METHOD bitXIsEqualTo
VAR_INPUT
	(* current value to check *)
	currentValue	:WORD;
	(* number of bit to check *)
	number			:BitNumberWord;
	(* expected value of bit *)
	expectedValue	:BOOL;
	(* message if the assertion is false *)
	message			:AssertMessage;
END_VAR
IF (
	TO_BOOL(
		TO_WORD(SHL(THIS^.LSB, number))
		AND currentValue
	) <> expectedValue
) THEN
	THIS^.assertionWasWrong(message, THIS^.getDebugInfo('bitXIsEqualTo'));
END_IF
END_METHOD

(*

short summary
=================
This assertion method checks if the selected bit of current value
is not equal to the unexpected value

.. <legal notes>

legal notes
=================
| SPDX-FileCopyrightText: © 2022 ekvip automation GmbH <info@ekvip.de>
| SPDX-License-Identifier: Apache-2.0
| For details check: Apache-2.0_

.. _Apache-2.0: https://www.apache.org/licenses/LICENSE-2.0

.. </legal notes>

parameters
=================

*)

METHOD bitXIsNotEqualTo
VAR_INPUT
	(* current value to check *)
	currentValue	:WORD;
	(* number of bit to check *)
	number			:BitNumberWord;
	(* unexpected value of bit *)
	unexpectedValue	:BOOL;
	(* message if the assertion is false *)
	message			:AssertMessage;
END_VAR
IF (
	TO_BOOL(
		TO_WORD(SHL(THIS^.LSB, number))
		AND currentValue
	) = unexpectedValue
) THEN
	THIS^.assertionWasWrong(message, THIS^.getDebugInfo('bitXIsNotEqualTo'));
END_IF
END_METHOD

(*

short summary
=================
This assertion method checks if the selected bit of current value
is set

.. <legal notes>

legal notes
=================
| SPDX-FileCopyrightText: © 2022 ekvip automation GmbH <info@ekvip.de>
| SPDX-License-Identifier: Apache-2.0
| For details check: Apache-2.0_

.. _Apache-2.0: https://www.apache.org/licenses/LICENSE-2.0

.. </legal notes>

parameters
=================

*)

METHOD bitXIsSet
VAR_INPUT
	(* current value to check *)
	currentValue	:WORD;
	(* number of bit to check *)
	number			:BitNumberWord;
	(* message if the assertion is false *)
	message			:AssertMessage;
END_VAR
IF (
	NOT TO_BOOL(
		TO_WORD(SHL(THIS^.LSB, number))
		AND currentValue
	)
) THEN
	THIS^.assertionWasWrong(message, THIS^.getDebugInfo('bitXIsSet'));
END_IF
END_METHOD

(*

short summary
=================
This assertion method checks if the selected bit of current value
is unset

.. <legal notes>

legal notes
=================
| SPDX-FileCopyrightText: © 2022 ekvip automation GmbH <info@ekvip.de>
| SPDX-License-Identifier: Apache-2.0
| For details check: Apache-2.0_

.. _Apache-2.0: https://www.apache.org/licenses/LICENSE-2.0

.. </legal notes>

parameters
=================

*)

METHOD bitXIsUnset
VAR_INPUT
	(* current value to check *)
	currentValue	:WORD;
	(* number of bit to check *)
	number			:BitNumberWord;
	(* message if the assertion is false *)
	message			:AssertMessage;
END_VAR
IF (
	TO_BOOL(
		TO_WORD(SHL(THIS^.LSB, number))
		AND currentValue
	)
) THEN
	THIS^.assertionWasWrong(message, THIS^.getDebugInfo('bitXIsUnset'));
END_IF
END_METHOD

(*

short summary
=================
This abstract property returns the class name of the concrete object, 
It's for debugging purpose

.. <legal notes>

legal notes
=================
| SPDX-FileCopyrightText: © 2022 ekvip automation GmbH <info@ekvip.de>
| SPDX-License-Identifier: Apache-2.0
| For details check: Apache-2.0_

.. _Apache-2.0: https://www.apache.org/licenses/LICENSE-2.0

.. </legal notes>

*)

PROPERTY className :CNM_AbstractObject.ClassName
GET
className := 'CNM_AssertionInterfaceLib.WordAssertions';
END_GET
END_PROPERTY

(*

short summary
=================
This assertion method checks if the least significant bit of current value
is equal to the expected value

.. <legal notes>

legal notes
=================
| SPDX-FileCopyrightText: © 2022 ekvip automation GmbH <info@ekvip.de>
| SPDX-License-Identifier: Apache-2.0
| For details check: Apache-2.0_

.. _Apache-2.0: https://www.apache.org/licenses/LICENSE-2.0

.. </legal notes>

parameters
=================

*)

METHOD lsbIsEqualTo
VAR_INPUT
	(* current value to check *)
	currentValue	:WORD;
	(* expected value of lsb *)
	expectedValue	:BOOL;
	(* message if the assertion is false *)
	message			:AssertMessage;
END_VAR
IF (TO_BOOL(currentValue AND THIS^.LSB) <> expectedValue) THEN
	THIS^.assertionWasWrong(message, THIS^.getDebugInfo('lsbIsEqualTo'));
END_IF
END_METHOD

(*

short summary
=================
This assertion method checks if the least significant bit of current value
is not equal to the unexpected value

.. <legal notes>

legal notes
=================
| SPDX-FileCopyrightText: © 2022 ekvip automation GmbH <info@ekvip.de>
| SPDX-License-Identifier: Apache-2.0
| For details check: Apache-2.0_

.. _Apache-2.0: https://www.apache.org/licenses/LICENSE-2.0

.. </legal notes>

parameters
=================

*)

METHOD lsbIsNotEqualTo
VAR_INPUT
	(* current value to check *)
	currentValue	:WORD;
	(* unexpected value of lsb *)
	unexpectedValue	:BOOL;
	(* message if the assertion is false *)
	message			:AssertMessage;
END_VAR
IF (TO_BOOL(currentValue AND THIS^.LSB) = unexpectedValue) THEN
	THIS^.assertionWasWrong(message, THIS^.getDebugInfo('lsbIsNotEqualTo'));
END_IF
END_METHOD

(*

short summary
=================
This assertion method checks if the least significant bit of current value
is set

.. <legal notes>

legal notes
=================
| SPDX-FileCopyrightText: © 2022 ekvip automation GmbH <info@ekvip.de>
| SPDX-License-Identifier: Apache-2.0
| For details check: Apache-2.0_

.. _Apache-2.0: https://www.apache.org/licenses/LICENSE-2.0

.. </legal notes>

parameters
=================

*)

METHOD lsbIsSet
VAR_INPUT
	(* current value to check *)
	currentValue	:WORD;
	(* message if the assertion is false *)
	message			:AssertMessage;
END_VAR
IF (NOT TO_BOOL(currentValue AND THIS^.LSB)) THEN
	THIS^.assertionWasWrong(message, THIS^.getDebugInfo('lsbIsSet'));
END_IF
END_METHOD

(*

short summary
=================
This assertion method checks if the least significant bit of current value
is unset

.. <legal notes>

legal notes
=================
| SPDX-FileCopyrightText: © 2022 ekvip automation GmbH <info@ekvip.de>
| SPDX-License-Identifier: Apache-2.0
| For details check: Apache-2.0_

.. _Apache-2.0: https://www.apache.org/licenses/LICENSE-2.0

.. </legal notes>

parameters
=================

*)

METHOD lsbIsUnset
VAR_INPUT
	(* current value to check *)
	currentValue	:WORD;
	(* message if the assertion is false *)
	message			:AssertMessage;
END_VAR
IF (TO_BOOL(currentValue AND THIS^.LSB)) THEN
	THIS^.assertionWasWrong(message, THIS^.getDebugInfo('lsbIsUnset'));
END_IF
END_METHOD

(*

short summary
=================
This assertion method checks if the most significant bit of current value
is equal to the expected value

.. <legal notes>

legal notes
=================
| SPDX-FileCopyrightText: © 2022 ekvip automation GmbH <info@ekvip.de>
| SPDX-License-Identifier: Apache-2.0
| For details check: Apache-2.0_

.. _Apache-2.0: https://www.apache.org/licenses/LICENSE-2.0

.. </legal notes>

parameters
=================

*)

METHOD msbIsEqualTo
VAR_INPUT
	(* current value to check *)
	currentValue	:WORD;
	(* expected value of msb *)
	expectedValue	:BOOL;
	(* message if the assertion is false *)
	message			:AssertMessage;
END_VAR
IF (TO_BOOL(currentValue AND THIS^.MSB) <> expectedValue) THEN
	THIS^.assertionWasWrong(message, THIS^.getDebugInfo('msbIsEqualTo'));
END_IF
END_METHOD

(*

short summary
=================
This assertion method checks if the most significant bit of current value
is not equal to the unexpected value

.. <legal notes>

legal notes
=================
| SPDX-FileCopyrightText: © 2022 ekvip automation GmbH <info@ekvip.de>
| SPDX-License-Identifier: Apache-2.0
| For details check: Apache-2.0_

.. _Apache-2.0: https://www.apache.org/licenses/LICENSE-2.0

.. </legal notes>

parameters
=================

*)

METHOD msbIsNotEqualTo
VAR_INPUT
	(* current value to check *)
	currentValue	:WORD;
	(* unexpected value of msb *)
	unexpectedValue	:BOOL;
	(* message if the assertion is false *)
	message			:AssertMessage;
END_VAR
IF (TO_BOOL(currentValue AND THIS^.MSB) = unexpectedValue) THEN
	THIS^.assertionWasWrong(message, THIS^.getDebugInfo('msbIsNotEqualTo'));
END_IF
END_METHOD

(*

short summary
=================
This assertion method checks if the most significant bit of current value
is set

.. <legal notes>

legal notes
=================
| SPDX-FileCopyrightText: © 2022 ekvip automation GmbH <info@ekvip.de>
| SPDX-License-Identifier: Apache-2.0
| For details check: Apache-2.0_

.. _Apache-2.0: https://www.apache.org/licenses/LICENSE-2.0

.. </legal notes>

parameters
=================

*)

METHOD msbIsSet
VAR_INPUT
	(* current value to check *)
	currentValue	:WORD;
	(* message if the assertion is false *)
	message			:AssertMessage;
END_VAR
IF (NOT TO_BOOL(currentValue AND THIS^.MSB)) THEN
	THIS^.assertionWasWrong(message, THIS^.getDebugInfo('msbIsSet'));
END_IF
END_METHOD

(*

short summary
=================
This assertion method checks if the most significant bit of current value
is unset

.. <legal notes>

legal notes
=================
| SPDX-FileCopyrightText: © 2022 ekvip automation GmbH <info@ekvip.de>
| SPDX-License-Identifier: Apache-2.0
| For details check: Apache-2.0_

.. _Apache-2.0: https://www.apache.org/licenses/LICENSE-2.0

.. </legal notes>

parameters
=================

*)

METHOD msbIsUnset
VAR_INPUT
	(* current value to check *)
	currentValue	:WORD;
	(* message if the assertion is false *)
	message			:AssertMessage;
END_VAR
IF (TO_BOOL(currentValue AND THIS^.MSB)) THEN
	THIS^.assertionWasWrong(message, THIS^.getDebugInfo('msbIsUnset'));
END_IF
END_METHOD

(*

short summary
=================
This assertion method checks if the result current value bitwise ``OR`` mask is equal to the expected value

.. <legal notes>

legal notes
=================
| SPDX-FileCopyrightText: © 2022 ekvip automation GmbH <info@ekvip.de>
| SPDX-License-Identifier: Apache-2.0
| For details check: Apache-2.0_

.. _Apache-2.0: https://www.apache.org/licenses/LICENSE-2.0

.. </legal notes>

parameters
=================

*)

METHOD orMaskIsEqualTo
VAR_INPUT
	(* current value to check *)
	currentValue	:WORD;
	(* 2nd operand for bitwise operation *)
	mask			:WORD;
	(* expected result after masking *)
	expectedValue	:WORD;
	(* message if the assertion is false *)
	message			:AssertMessage;
END_VAR
IF ((currentValue OR mask) <> expectedValue) THEN
	THIS^.assertionWasWrong(message, THIS^.getDebugInfo('orMaskIsEqualTo'));
END_IF
END_METHOD

(*

short summary
=================
This assertion method checks if the result current value bitwise ``OR`` mask 
is not equal to the unexpected value

.. <legal notes>

legal notes
=================
| SPDX-FileCopyrightText: © 2022 ekvip automation GmbH <info@ekvip.de>
| SPDX-License-Identifier: Apache-2.0
| For details check: Apache-2.0_

.. _Apache-2.0: https://www.apache.org/licenses/LICENSE-2.0

.. </legal notes>

parameters
=================

*)

METHOD orMaskIsNotEqualTo
VAR_INPUT
	(* current value to check *)
	currentValue	:WORD;
	(* 2nd operand for bitwise operation *)
	mask			:WORD;
	(* unexpected result after masking *)
	unexpectedValue	:WORD;
	(* message if the assertion is false *)
	message			:AssertMessage;
END_VAR
IF ((currentValue OR mask) = unexpectedValue) THEN
	THIS^.assertionWasWrong(message, THIS^.getDebugInfo('orMaskIsNotEqualTo'));
END_IF
END_METHOD

(*

short summary
=================
This assertion method checks if the current value is equal to the expected value

.. <legal notes>

legal notes
=================
| SPDX-FileCopyrightText: © 2022 ekvip automation GmbH <info@ekvip.de>
| SPDX-License-Identifier: Apache-2.0
| For details check: Apache-2.0_

.. _Apache-2.0: https://www.apache.org/licenses/LICENSE-2.0

.. </legal notes>

parameters
=================

*)

METHOD valueIsEqualTo
VAR_INPUT
	(* current value to check *)
	currentValue	:WORD;
	(* expected value to compare *)
	expectedValue	:WORD;
	(* message if the assertion is false *)
	message			:AssertMessage;
END_VAR
IF (currentValue <> expectedValue) THEN
	THIS^.assertionWasWrong(message, THIS^.getDebugInfo('valueIsEqualTo'));
END_IF
END_METHOD

(*

short summary
=================
This assertion method checks if the current value is greater than the less value

.. <legal notes>

legal notes
=================
| SPDX-FileCopyrightText: © 2022 ekvip automation GmbH <info@ekvip.de>
| SPDX-License-Identifier: Apache-2.0
| For details check: Apache-2.0_

.. _Apache-2.0: https://www.apache.org/licenses/LICENSE-2.0

.. </legal notes>

parameters
=================

*)

METHOD valueIsGreaterThan
VAR_INPUT
	(* current value to check *)
	currentValue	:WORD;
	(* less than lower limit *)
	lessValue		:WORD;
	(* message if the assertion is false *)
	message			:AssertMessage;
END_VAR
IF (currentValue <= lessValue) THEN
	THIS^.assertionWasWrong(message, THIS^.getDebugInfo('valueIsGreaterThan'));
END_IF
END_METHOD

(*

short summary
=================
This assertion method checks if the current value is inside a limit

.. attention:: 
	limits are included: ``valueIsInRangeOf(3, 3, 3)`` is a true assertion

.. <legal notes>

legal notes
=================
| SPDX-FileCopyrightText: © 2022 ekvip automation GmbH <info@ekvip.de>
| SPDX-License-Identifier: Apache-2.0
| For details check: Apache-2.0_

.. _Apache-2.0: https://www.apache.org/licenses/LICENSE-2.0

.. </legal notes>

parameters
=================

*)

METHOD valueIsInRangeOf
VAR_INPUT
	(* lower limit for the current value *)
	lowerLimit		:WORD;
	(* current value to check *)
	currentValue	:WORD;
	(* upper limit for the current value *)
	upperLimit		:WORD;
	(* message if the assertion is false *)
	message			:AssertMessage;
END_VAR
IF (
	(currentValue < lowerLimit)
	OR (currentValue > upperLimit)
) THEN
	THIS^.assertionWasWrong(message, THIS^.getDebugInfo('valueIsInRangeOf'));
END_IF
END_METHOD

(*

short summary
=================
This assertion method checks if the current value is less than the greater value

.. <legal notes>

legal notes
=================
| SPDX-FileCopyrightText: © 2022 ekvip automation GmbH <info@ekvip.de>
| SPDX-License-Identifier: Apache-2.0
| For details check: Apache-2.0_

.. _Apache-2.0: https://www.apache.org/licenses/LICENSE-2.0

.. </legal notes>

parameters
=================

*)

METHOD valueIsLessThan
VAR_INPUT
	(* current value to check *)
	currentValue	:WORD;
	(* greater than upper limit *)
	greaterValue	:WORD;
	(* message if the assertion is false *)
	message			:AssertMessage;
END_VAR
IF (currentValue >= greaterValue) THEN
	THIS^.assertionWasWrong(message, THIS^.getDebugInfo('valueIsLessThan'));
END_IF
END_METHOD

(*

short summary
=================
This assertion method checks if the current value is less than or equal to the maximum value

.. <legal notes>

legal notes
=================
| SPDX-FileCopyrightText: © 2022 ekvip automation GmbH <info@ekvip.de>
| SPDX-License-Identifier: Apache-2.0
| For details check: Apache-2.0_

.. _Apache-2.0: https://www.apache.org/licenses/LICENSE-2.0

.. </legal notes>

parameters
=================

*)

METHOD valueIsMax
VAR_INPUT
	(* current value to check *)
	currentValue	:WORD;
	(* upper limit for the current value *)
	maximumValue	:WORD;
	(* message if the assertion is false *)
	message			:AssertMessage;
END_VAR
IF (currentValue > maximumValue) THEN
	THIS^.assertionWasWrong(message, THIS^.getDebugInfo('valueIsMax'));
END_IF
END_METHOD

(*

short summary
=================
This assertion method checks if the current value is greater than or equal to the minimum value

.. <legal notes>

legal notes
=================
| SPDX-FileCopyrightText: © 2022 ekvip automation GmbH <info@ekvip.de>
| SPDX-License-Identifier: Apache-2.0
| For details check: Apache-2.0_

.. _Apache-2.0: https://www.apache.org/licenses/LICENSE-2.0

.. </legal notes>

parameters
=================

*)

METHOD valueIsMin
VAR_INPUT
	(* current value to check *)
	currentValue	:WORD;
	(* lower limit for the current value *)
	minimumValue	:WORD;
	(* message if the assertion is false *)
	message			:AssertMessage;
END_VAR
IF (currentValue < minimumValue) THEN
	THIS^.assertionWasWrong(message, THIS^.getDebugInfo('valueIsMin'));
END_IF
END_METHOD

(*

short summary
=================
This assertion method checks if the current value is not equal to the unexpected value

.. <legal notes>

legal notes
=================
| SPDX-FileCopyrightText: © 2022 ekvip automation GmbH <info@ekvip.de>
| SPDX-License-Identifier: Apache-2.0
| For details check: Apache-2.0_

.. _Apache-2.0: https://www.apache.org/licenses/LICENSE-2.0

.. </legal notes>

parameters
=================

*)

METHOD valueIsNotEqualTo
VAR_INPUT
	(* current value to check *)
	currentValue	:WORD;
	(* unexpected value to compare *)
	unexpectedValue	:WORD;
	(* message if the assertion is false *)
	message			:AssertMessage;
END_VAR
IF (currentValue = unexpectedValue) THEN
	THIS^.assertionWasWrong(message, THIS^.getDebugInfo('valueIsNotEqualTo'));
END_IF
END_METHOD

(*

short summary
=================
This assertion method checks if the result current value bitwise ``XOR`` mask is equal to the expected value

.. <legal notes>

legal notes
=================
| SPDX-FileCopyrightText: © 2022 ekvip automation GmbH <info@ekvip.de>
| SPDX-License-Identifier: Apache-2.0
| For details check: Apache-2.0_

.. _Apache-2.0: https://www.apache.org/licenses/LICENSE-2.0

.. </legal notes>

parameters
=================

*)

METHOD xorMaskIsEqualTo
VAR_INPUT
	(* current value to check *)
	currentValue	:WORD;
	(* 2nd operand for bitwise operation *)
	mask			:WORD;
	(* expected result after masking *)
	expectedValue	:WORD;
	(* message if the assertion is false *)
	message			:AssertMessage;
END_VAR
IF ((currentValue XOR mask) <> expectedValue) THEN
	THIS^.assertionWasWrong(message, THIS^.getDebugInfo('xorMaskIsEqualTo'));
END_IF
END_METHOD

(*

short summary
=================
This assertion method checks if the result current value bitwise ``XOR`` mask 
is not equal to the unexpected value

.. <legal notes>

legal notes
=================
| SPDX-FileCopyrightText: © 2022 ekvip automation GmbH <info@ekvip.de>
| SPDX-License-Identifier: Apache-2.0
| For details check: Apache-2.0_

.. _Apache-2.0: https://www.apache.org/licenses/LICENSE-2.0

.. </legal notes>

parameters
=================

*)

METHOD xorMaskIsNotEqualTo
VAR_INPUT
	(* current value to check *)
	currentValue	:WORD;
	(* 2nd operand for bitwise operation *)
	mask			:WORD;
	(* unexpected result after masking *)
	unexpectedValue	:WORD;
	(* message if the assertion is false *)
	message			:AssertMessage;
END_VAR
IF ((currentValue XOR mask) = unexpectedValue) THEN
	THIS^.assertionWasWrong(message, THIS^.getDebugInfo('xorMaskIsNotEqualTo'));
END_IF
END_METHOD

END_FUNCTION_BLOCK

// ---- Assertor/Assertions/BitNumberAssertions/Dword/classes/DWordAssertions.TcPOU
(*

short summary
=================
This class provides assert statements for double words  
It implements :ref:`IDWordAssertions`

.. <legal notes>

legal notes
=================
| SPDX-FileCopyrightText: © 2022 ekvip automation GmbH <info@ekvip.de>
| SPDX-License-Identifier: Apache-2.0
| For details check: Apache-2.0_

.. _Apache-2.0: https://www.apache.org/licenses/LICENSE-2.0

.. </legal notes>

methods and properties
=======================

*)

{attribute 'reflection'}
FUNCTION_BLOCK INTERNAL DWordAssertions EXTENDS AbstactAssertion IMPLEMENTS IDWordAssertions
VAR
END_VAR
VAR CONSTANT
	(* least significant bit *)
	LSB	:DWORD := 16#0000_0001;
	(* most significant bit *)
	MSB :DWORD := 16#8000_0000;
END_VAR

(*

short summary
=================
This assertion method checks if the result current value bitwise ``AND`` mask is equal to the expected value

.. <legal notes>

legal notes
=================
| SPDX-FileCopyrightText: © 2022 ekvip automation GmbH <info@ekvip.de>
| SPDX-License-Identifier: Apache-2.0
| For details check: Apache-2.0_

.. _Apache-2.0: https://www.apache.org/licenses/LICENSE-2.0

.. </legal notes>

parameters
=================

*)

METHOD andMaskIsEqualTo
VAR_INPUT
	(* current value to check *)
	currentValue	:DWORD;
	(* 2nd operand for bitwise operation *)
	mask			:DWORD;
	(* expected result after masking *)
	expectedValue	:DWORD;
	(* message if the assertion is false *)
	message			:AssertMessage;
END_VAR
IF ((currentValue AND mask) <> expectedValue) THEN
	THIS^.assertionWasWrong(message, THIS^.getDebugInfo('andMaskIsEqualTo'));
END_IF
END_METHOD

(*

short summary
=================
This assertion method checks if the result current value bitwise ``AND`` mask
is not equal to the unexpected value

.. <legal notes>

legal notes
=================
| SPDX-FileCopyrightText: © 2022 ekvip automation GmbH <info@ekvip.de>
| SPDX-License-Identifier: Apache-2.0
| For details check: Apache-2.0_

.. _Apache-2.0: https://www.apache.org/licenses/LICENSE-2.0

.. </legal notes>

parameters
=================

*)

METHOD andMaskIsNotEqualTo
VAR_INPUT
	(* current value to check *)
	currentValue	:DWORD;
	(* 2nd operand for bitwise operation *)
	mask			:DWORD;
	(* unexpected result after masking *)
	unexpectedValue	:DWORD;
	(* message if the assertion is false *)
	message			:AssertMessage;
END_VAR
IF ((currentValue AND mask) = unexpectedValue) THEN
	THIS^.assertionWasWrong(message, THIS^.getDebugInfo('andMaskIsNotEqualTo'));
END_IF
END_METHOD

(*

short summary
=================
This assertion method checks if the selected bit of current value
is equal to the expected value

.. <legal notes>

legal notes
=================
| SPDX-FileCopyrightText: © 2022 ekvip automation GmbH <info@ekvip.de>
| SPDX-License-Identifier: Apache-2.0
| For details check: Apache-2.0_

.. _Apache-2.0: https://www.apache.org/licenses/LICENSE-2.0

.. </legal notes>

parameters
=================

*)

METHOD bitXIsEqualTo
VAR_INPUT
	(* current value to check *)
	currentValue	:DWORD;
	(* number of bit to check *)
	number			:BitNumberDWord;
	(* expected value of bit *)
	expectedValue	:BOOL;
	(* message if the assertion is false *)
	message			:AssertMessage;
END_VAR
IF (
	TO_BOOL(
		TO_DWORD(SHL(THIS^.LSB, number))
		AND currentValue
	) <> expectedValue
) THEN
	THIS^.assertionWasWrong(message, THIS^.getDebugInfo('bitXIsEqualTo'));
END_IF
END_METHOD

(*

short summary
=================
This assertion method checks if the selected bit of current value
is not equal to the unexpected value

.. <legal notes>

legal notes
=================
| SPDX-FileCopyrightText: © 2022 ekvip automation GmbH <info@ekvip.de>
| SPDX-License-Identifier: Apache-2.0
| For details check: Apache-2.0_

.. _Apache-2.0: https://www.apache.org/licenses/LICENSE-2.0

.. </legal notes>

parameters
=================

*)

METHOD bitXIsNotEqualTo
VAR_INPUT
	(* current value to check *)
	currentValue	:DWORD;
	(* number of bit to check *)
	number			:BitNumberDWord;
	(* unexpected value of bit *)
	unexpectedValue	:BOOL;
	(* message if the assertion is false *)
	message			:AssertMessage;
END_VAR
IF (
	TO_BOOL(
		TO_DWORD(SHL(THIS^.LSB, number))
		AND currentValue
	) = unexpectedValue
) THEN
	THIS^.assertionWasWrong(message, THIS^.getDebugInfo('bitXIsNotEqualTo'));
END_IF
END_METHOD

(*

short summary
=================
This assertion method checks if the selected bit of current value
is set

.. <legal notes>

legal notes
=================
| SPDX-FileCopyrightText: © 2022 ekvip automation GmbH <info@ekvip.de>
| SPDX-License-Identifier: Apache-2.0
| For details check: Apache-2.0_

.. _Apache-2.0: https://www.apache.org/licenses/LICENSE-2.0

.. </legal notes>

parameters
=================

*)

METHOD bitXIsSet
VAR_INPUT
	(* current value to check *)
	currentValue	:DWORD;
	(* number of bit to check *)
	number			:BitNumberDWord;
	(* message if the assertion is false *)
	message			:AssertMessage;
END_VAR
IF (
	NOT TO_BOOL(
		TO_DWORD(SHL(THIS^.LSB, number))
		AND currentValue
	)
) THEN
	THIS^.assertionWasWrong(message, THIS^.getDebugInfo('bitXIsSet'));
END_IF
END_METHOD

(*

short summary
=================
This assertion method checks if the selected bit of current value
is unset

.. <legal notes>

legal notes
=================
| SPDX-FileCopyrightText: © 2022 ekvip automation GmbH <info@ekvip.de>
| SPDX-License-Identifier: Apache-2.0
| For details check: Apache-2.0_

.. _Apache-2.0: https://www.apache.org/licenses/LICENSE-2.0

.. </legal notes>

parameters
=================

*)

METHOD bitXIsUnset
VAR_INPUT
	(* current value to check *)
	currentValue	:DWORD;
	(* number of bit to check *)
	number			:BitNumberDWord;
	(* message if the assertion is false *)
	message			:AssertMessage;
END_VAR
IF (
	TO_BOOL(
		TO_DWORD(SHL(THIS^.LSB, number))
		AND currentValue
	)
) THEN
	THIS^.assertionWasWrong(message, THIS^.getDebugInfo('bitXIsUnset'));
END_IF
END_METHOD

(*

short summary
=================
This abstract property returns the class name of the concrete object, 
It's for debugging purpose

.. <legal notes>

legal notes
=================
| SPDX-FileCopyrightText: © 2022 ekvip automation GmbH <info@ekvip.de>
| SPDX-License-Identifier: Apache-2.0
| For details check: Apache-2.0_

.. _Apache-2.0: https://www.apache.org/licenses/LICENSE-2.0

.. </legal notes>

*)

PROPERTY className :CNM_AbstractObject.ClassName
GET
className := 'CNM_AssertionInterfaceLib.DWordAssertions';
END_GET
END_PROPERTY

(*

short summary
=================
This assertion method checks if the least significant bit of current value
is equal to the expected value

.. <legal notes>

legal notes
=================
| SPDX-FileCopyrightText: © 2022 ekvip automation GmbH <info@ekvip.de>
| SPDX-License-Identifier: Apache-2.0
| For details check: Apache-2.0_

.. _Apache-2.0: https://www.apache.org/licenses/LICENSE-2.0

.. </legal notes>

parameters
=================

*)

METHOD lsbIsEqualTo
VAR_INPUT
	(* current value to check *)
	currentValue	:DWORD;
	(* expected value of lsb *)
	expectedValue	:BOOL;
	(* message if the assertion is false *)
	message			:AssertMessage;
END_VAR
IF (TO_BOOL(currentValue AND THIS^.LSB) <> expectedValue) THEN
	THIS^.assertionWasWrong(message, THIS^.getDebugInfo('lsbIsEqualTo'));
END_IF
END_METHOD

(*

short summary
=================
This assertion method checks if the least significant bit of current value
is not equal to the unexpected value

.. <legal notes>

legal notes
=================
| SPDX-FileCopyrightText: © 2022 ekvip automation GmbH <info@ekvip.de>
| SPDX-License-Identifier: Apache-2.0
| For details check: Apache-2.0_

.. _Apache-2.0: https://www.apache.org/licenses/LICENSE-2.0

.. </legal notes>

parameters
=================

*)

METHOD lsbIsNotEqualTo
VAR_INPUT
	(* current value to check *)
	currentValue	:DWORD;
	(* unexpected value of lsb *)
	unexpectedValue	:BOOL;
	(* message if the assertion is false *)
	message			:AssertMessage;
END_VAR
IF (TO_BOOL(currentValue AND THIS^.LSB) = unexpectedValue) THEN
	THIS^.assertionWasWrong(message, THIS^.getDebugInfo('lsbIsNotEqualTo'));
END_IF
END_METHOD

(*

short summary
=================
This assertion method checks if the least significant bit of current value
is set

.. <legal notes>

legal notes
=================
| SPDX-FileCopyrightText: © 2022 ekvip automation GmbH <info@ekvip.de>
| SPDX-License-Identifier: Apache-2.0
| For details check: Apache-2.0_

.. _Apache-2.0: https://www.apache.org/licenses/LICENSE-2.0

.. </legal notes>

parameters
=================

*)

METHOD lsbIsSet
VAR_INPUT
	(* current value to check *)
	currentValue	:DWORD;
	(* message if the assertion is false *)
	message			:AssertMessage;
END_VAR
IF (NOT TO_BOOL(currentValue AND THIS^.LSB)) THEN
	THIS^.assertionWasWrong(message, THIS^.getDebugInfo('lsbIsSet'));
END_IF
END_METHOD

(*

short summary
=================
This assertion method checks if the least significant bit of current value
is unset

.. <legal notes>

legal notes
=================
| SPDX-FileCopyrightText: © 2022 ekvip automation GmbH <info@ekvip.de>
| SPDX-License-Identifier: Apache-2.0
| For details check: Apache-2.0_

.. _Apache-2.0: https://www.apache.org/licenses/LICENSE-2.0

.. </legal notes>

parameters
=================

*)

METHOD lsbIsUnset
VAR_INPUT
	(* current value to check *)
	currentValue	:DWORD;
	(* message if the assertion is false *)
	message			:AssertMessage;
END_VAR
IF (TO_BOOL(currentValue AND THIS^.LSB)) THEN
	THIS^.assertionWasWrong(message, THIS^.getDebugInfo('lsbIsUnset'));
END_IF
END_METHOD

(*

short summary
=================
This assertion method checks if the most significant bit of current value
is equal to the expected value

.. <legal notes>

legal notes
=================
| SPDX-FileCopyrightText: © 2022 ekvip automation GmbH <info@ekvip.de>
| SPDX-License-Identifier: Apache-2.0
| For details check: Apache-2.0_

.. _Apache-2.0: https://www.apache.org/licenses/LICENSE-2.0

.. </legal notes>

parameters
=================

*)

METHOD msbIsEqualTo
VAR_INPUT
	(* current value to check *)
	currentValue	:DWORD;
	(* expected value of msb *)
	expectedValue	:BOOL;
	(* message if the assertion is false *)
	message			:AssertMessage;
END_VAR
IF (TO_BOOL(currentValue AND THIS^.MSB) <> expectedValue) THEN
	THIS^.assertionWasWrong(message, THIS^.getDebugInfo('msbIsEqualTo'));
END_IF
END_METHOD

(*

short summary
=================
This assertion method checks if the most significant bit of current value
is not equal to the unexpected value

.. <legal notes>

legal notes
=================
| SPDX-FileCopyrightText: © 2022 ekvip automation GmbH <info@ekvip.de>
| SPDX-License-Identifier: Apache-2.0
| For details check: Apache-2.0_

.. _Apache-2.0: https://www.apache.org/licenses/LICENSE-2.0

.. </legal notes>

parameters
=================

*)

METHOD msbIsNotEqualTo
VAR_INPUT
	(* current value to check *)
	currentValue	:DWORD;
	(* unexpected value of msb *)
	unexpectedValue	:BOOL;
	(* message if the assertion is false *)
	message			:AssertMessage;
END_VAR
IF (TO_BOOL(currentValue AND THIS^.MSB) = unexpectedValue) THEN
	THIS^.assertionWasWrong(message, THIS^.getDebugInfo('msbIsNotEqualTo'));
END_IF
END_METHOD

(*

short summary
=================
This assertion method checks if the most significant bit of current value
is set

.. <legal notes>

legal notes
=================
| SPDX-FileCopyrightText: © 2022 ekvip automation GmbH <info@ekvip.de>
| SPDX-License-Identifier: Apache-2.0
| For details check: Apache-2.0_

.. _Apache-2.0: https://www.apache.org/licenses/LICENSE-2.0

.. </legal notes>

parameters
=================

*)

METHOD msbIsSet
VAR_INPUT
	(* current value to check *)
	currentValue	:DWORD;
	(* message if the assertion is false *)
	message			:AssertMessage;
END_VAR
IF (NOT TO_BOOL(currentValue AND THIS^.MSB)) THEN
	THIS^.assertionWasWrong(message, THIS^.getDebugInfo('msbIsSet'));
END_IF
END_METHOD

(*

short summary
=================
This assertion method checks if the most significant bit of current value
is unset

.. <legal notes>

legal notes
=================
| SPDX-FileCopyrightText: © 2022 ekvip automation GmbH <info@ekvip.de>
| SPDX-License-Identifier: Apache-2.0
| For details check: Apache-2.0_

.. _Apache-2.0: https://www.apache.org/licenses/LICENSE-2.0

.. </legal notes>

parameters
=================

*)

METHOD msbIsUnset
VAR_INPUT
	(* current value to check *)
	currentValue	:DWORD;
	(* message if the assertion is false *)
	message			:AssertMessage;
END_VAR
IF (TO_BOOL(currentValue AND THIS^.MSB)) THEN
	THIS^.assertionWasWrong(message, THIS^.getDebugInfo('msbIsUnset'));
END_IF
END_METHOD

(*

short summary
=================
This assertion method checks if the result current value bitwise ``OR`` mask is equal to the expected value

.. <legal notes>

legal notes
=================
| SPDX-FileCopyrightText: © 2022 ekvip automation GmbH <info@ekvip.de>
| SPDX-License-Identifier: Apache-2.0
| For details check: Apache-2.0_

.. _Apache-2.0: https://www.apache.org/licenses/LICENSE-2.0

.. </legal notes>

parameters
=================

*)

METHOD orMaskIsEqualTo
VAR_INPUT
	(* current value to check *)
	currentValue	:DWORD;
	(* 2nd operand for bitwise operation *)
	mask			:DWORD;
	(* expected result after masking *)
	expectedValue	:DWORD;
	(* message if the assertion is false *)
	message			:AssertMessage;
END_VAR
IF ((currentValue OR mask) <> expectedValue) THEN
	THIS^.assertionWasWrong(message, THIS^.getDebugInfo('orMaskIsEqualTo'));
END_IF
END_METHOD

(*

short summary
=================
This assertion method checks if the result current value bitwise ``OR`` mask 
is not equal to the unexpected value

.. <legal notes>

legal notes
=================
| SPDX-FileCopyrightText: © 2022 ekvip automation GmbH <info@ekvip.de>
| SPDX-License-Identifier: Apache-2.0
| For details check: Apache-2.0_

.. _Apache-2.0: https://www.apache.org/licenses/LICENSE-2.0

.. </legal notes>

parameters
=================

*)

METHOD orMaskIsNotEqualTo
VAR_INPUT
	(* current value to check *)
	currentValue	:DWORD;
	(* 2nd operand for bitwise operation *)
	mask			:DWORD;
	(* unexpected result after masking *)
	unexpectedValue	:DWORD;
	(* message if the assertion is false *)
	message			:AssertMessage;
END_VAR
IF ((currentValue OR mask) = unexpectedValue) THEN
	THIS^.assertionWasWrong(message, THIS^.getDebugInfo('orMaskIsNotEqualTo'));
END_IF
END_METHOD

(*

short summary
=================
This assertion method checks if the current value is equal to the expected value

.. <legal notes>

legal notes
=================
| SPDX-FileCopyrightText: © 2022 ekvip automation GmbH <info@ekvip.de>
| SPDX-License-Identifier: Apache-2.0
| For details check: Apache-2.0_

.. _Apache-2.0: https://www.apache.org/licenses/LICENSE-2.0

.. </legal notes>

parameters
=================

*)

METHOD valueIsEqualTo
VAR_INPUT
	(* current value to check *)
	currentValue	:DWORD;
	(* expected value to compare *)
	expectedValue	:DWORD;
	(* message if the assertion is false *)
	message			:AssertMessage;
END_VAR
IF (currentValue <> expectedValue) THEN
	THIS^.assertionWasWrong(message, THIS^.getDebugInfo('valueIsEqualTo'));
END_IF
END_METHOD

(*

short summary
=================
This assertion method checks if the current value is greater than the less value

.. <legal notes>

legal notes
=================
| SPDX-FileCopyrightText: © 2022 ekvip automation GmbH <info@ekvip.de>
| SPDX-License-Identifier: Apache-2.0
| For details check: Apache-2.0_

.. _Apache-2.0: https://www.apache.org/licenses/LICENSE-2.0

.. </legal notes>

parameters
=================

*)

METHOD valueIsGreaterThan
VAR_INPUT
	(* current value to check *)
	currentValue	:DWORD;
	(* less than lower limit *)
	lessValue		:DWORD;
	(* message if the assertion is false *)
	message			:AssertMessage;
END_VAR
IF (currentValue <= lessValue) THEN
	THIS^.assertionWasWrong(message, THIS^.getDebugInfo('valueIsGreaterThan'));
END_IF
END_METHOD

(*

short summary
=================
This assertion method checks if the current value is inside a limit

.. attention:: 
	limits are included: ``valueIsInRangeOf(3, 3, 3)`` is a true assertion

.. <legal notes>

legal notes
=================
| SPDX-FileCopyrightText: © 2022 ekvip automation GmbH <info@ekvip.de>
| SPDX-License-Identifier: Apache-2.0
| For details check: Apache-2.0_

.. _Apache-2.0: https://www.apache.org/licenses/LICENSE-2.0

.. </legal notes>

parameters
=================

*)

METHOD valueIsInRangeOf
VAR_INPUT
	(* lower limit for the current value *)
	lowerLimit		:DWORD;
	(* current value to check *)
	currentValue	:DWORD;
	(* upper limit for the current value *)
	upperLimit		:DWORD;
	(* message if the assertion is false *)
	message			:AssertMessage;
END_VAR
IF (
	(currentValue < lowerLimit)
	OR (currentValue > upperLimit)
) THEN
	THIS^.assertionWasWrong(message, THIS^.getDebugInfo('valueIsInRangeOf'));
END_IF
END_METHOD

(*

short summary
=================
This assertion method checks if the current value is less than the greater value

.. <legal notes>

legal notes
=================
| SPDX-FileCopyrightText: © 2022 ekvip automation GmbH <info@ekvip.de>
| SPDX-License-Identifier: Apache-2.0
| For details check: Apache-2.0_

.. _Apache-2.0: https://www.apache.org/licenses/LICENSE-2.0

.. </legal notes>

parameters
=================

*)

METHOD valueIsLessThan
VAR_INPUT
	(* current value to check *)
	currentValue	:DWORD;
	(* greater than upper limit *)
	greaterValue	:DWORD;
	(* message if the assertion is false *)
	message			:AssertMessage;
END_VAR
IF (currentValue >= greaterValue) THEN
	THIS^.assertionWasWrong(message, THIS^.getDebugInfo('valueIsLessThan'));
END_IF
END_METHOD

(*

short summary
=================
This assertion method checks if the current value is less than or equal to the maximum value

.. <legal notes>

legal notes
=================
| SPDX-FileCopyrightText: © 2022 ekvip automation GmbH <info@ekvip.de>
| SPDX-License-Identifier: Apache-2.0
| For details check: Apache-2.0_

.. _Apache-2.0: https://www.apache.org/licenses/LICENSE-2.0

.. </legal notes>

parameters
=================

*)

METHOD valueIsMax
VAR_INPUT
	(* current value to check *)
	currentValue	:DWORD;
	(* upper limit for the current value *)
	maximumValue	:DWORD;
	(* message if the assertion is false *)
	message			:AssertMessage;
END_VAR
IF (currentValue > maximumValue) THEN
	THIS^.assertionWasWrong(message, THIS^.getDebugInfo('valueIsMax'));
END_IF
END_METHOD

(*

short summary
=================
This assertion method checks if the current value is greater than or equal to the minimum value

.. <legal notes>

legal notes
=================
| SPDX-FileCopyrightText: © 2022 ekvip automation GmbH <info@ekvip.de>
| SPDX-License-Identifier: Apache-2.0
| For details check: Apache-2.0_

.. _Apache-2.0: https://www.apache.org/licenses/LICENSE-2.0

.. </legal notes>

parameters
=================

*)

METHOD valueIsMin
VAR_INPUT
	(* current value to check *)
	currentValue	:DWORD;
	(* lower limit for the current value *)
	minimumValue	:DWORD;
	(* message if the assertion is false *)
	message			:AssertMessage;
END_VAR
IF (currentValue < minimumValue) THEN
	THIS^.assertionWasWrong(message, THIS^.getDebugInfo('valueIsMin'));
END_IF
END_METHOD

(*

short summary
=================
This assertion method checks if the current value is not equal to the unexpected value

.. <legal notes>

legal notes
=================
| SPDX-FileCopyrightText: © 2022 ekvip automation GmbH <info@ekvip.de>
| SPDX-License-Identifier: Apache-2.0
| For details check: Apache-2.0_

.. _Apache-2.0: https://www.apache.org/licenses/LICENSE-2.0

.. </legal notes>

parameters
=================

*)

METHOD valueIsNotEqualTo
VAR_INPUT
	(* current value to check *)
	currentValue	:DWORD;
	(* unexpected value to compare *)
	unexpectedValue	:DWORD;
	(* message if the assertion is false *)
	message			:AssertMessage;
END_VAR
IF (currentValue = unexpectedValue) THEN
	THIS^.assertionWasWrong(message, THIS^.getDebugInfo('valueIsNotEqualTo'));
END_IF
END_METHOD

(*

short summary
=================
This assertion method checks if the result current value bitwise ``XOR`` mask is equal to the expected value

.. <legal notes>

legal notes
=================
| SPDX-FileCopyrightText: © 2022 ekvip automation GmbH <info@ekvip.de>
| SPDX-License-Identifier: Apache-2.0
| For details check: Apache-2.0_

.. _Apache-2.0: https://www.apache.org/licenses/LICENSE-2.0

.. </legal notes>

parameters
=================

*)

METHOD xorMaskIsEqualTo
VAR_INPUT
	(* current value to check *)
	currentValue	:DWORD;
	(* 2nd operand for bitwise operation *)
	mask			:DWORD;
	(* expected result after masking *)
	expectedValue	:DWORD;
	(* message if the assertion is false *)
	message			:AssertMessage;
END_VAR
IF ((currentValue XOR mask) <> expectedValue) THEN
	THIS^.assertionWasWrong(message, THIS^.getDebugInfo('xorMaskIsEqualTo'));
END_IF
END_METHOD

(*

short summary
=================
This assertion method checks if the result current value bitwise ``XOR`` mask 
is not equal to the unexpected value

.. <legal notes>

legal notes
=================
| SPDX-FileCopyrightText: © 2022 ekvip automation GmbH <info@ekvip.de>
| SPDX-License-Identifier: Apache-2.0
| For details check: Apache-2.0_

.. _Apache-2.0: https://www.apache.org/licenses/LICENSE-2.0

.. </legal notes>

parameters
=================

*)

METHOD xorMaskIsNotEqualTo
VAR_INPUT
	(* current value to check *)
	currentValue	:DWORD;
	(* 2nd operand for bitwise operation *)
	mask			:DWORD;
	(* unexpected result after masking *)
	unexpectedValue	:DWORD;
	(* message if the assertion is false *)
	message			:AssertMessage;
END_VAR
IF ((currentValue XOR mask) = unexpectedValue) THEN
	THIS^.assertionWasWrong(message, THIS^.getDebugInfo('xorMaskIsNotEqualTo'));
END_IF
END_METHOD

END_FUNCTION_BLOCK

// ---- Assertor/Assertions/BitNumberAssertions/Lword/classes/LWordAssertions.TcPOU
(*

short summary
=================
This class provides assert statements for long words  
It implements :ref:`ILWordAssertions`

.. <legal notes>

legal notes
=================
| SPDX-FileCopyrightText: © 2022 ekvip automation GmbH <info@ekvip.de>
| SPDX-License-Identifier: Apache-2.0
| For details check: Apache-2.0_

.. _Apache-2.0: https://www.apache.org/licenses/LICENSE-2.0

.. </legal notes>

methods and properties
=======================

*)

{attribute 'reflection'}
FUNCTION_BLOCK INTERNAL LWordAssertions EXTENDS AbstactAssertion IMPLEMENTS ILWordAssertions
VAR
END_VAR
VAR CONSTANT
	(* least significant bit *)
	LSB	:LWORD := 16#0000_0000_0000_0001;
	(* most significant bit *)
	MSB :LWORD := 16#8000_0000_0000_0000;
END_VAR

(*

short summary
=================
This assertion method checks if the result current value bitwise ``AND`` mask is equal to the expected value

.. <legal notes>

legal notes
=================
| SPDX-FileCopyrightText: © 2022 ekvip automation GmbH <info@ekvip.de>
| SPDX-License-Identifier: Apache-2.0
| For details check: Apache-2.0_

.. _Apache-2.0: https://www.apache.org/licenses/LICENSE-2.0

.. </legal notes>

parameters
=================

*)

METHOD andMaskIsEqualTo
VAR_INPUT
	(* current value to check *)
	currentValue	:LWORD;
	(* 2nd operand for bitwise operation *)
	mask			:LWORD;
	(* expected result after masking *)
	expectedValue	:LWORD;
	(* message if the assertion is false *)
	message			:AssertMessage;
END_VAR
IF ((currentValue AND mask) <> expectedValue) THEN
	THIS^.assertionWasWrong(message, THIS^.getDebugInfo('andMaskIsEqualTo'));
END_IF
END_METHOD

(*

short summary
=================
This assertion method checks if the result current value bitwise ``AND`` mask
is not equal to the unexpected value

.. <legal notes>

legal notes
=================
| SPDX-FileCopyrightText: © 2022 ekvip automation GmbH <info@ekvip.de>
| SPDX-License-Identifier: Apache-2.0
| For details check: Apache-2.0_

.. _Apache-2.0: https://www.apache.org/licenses/LICENSE-2.0

.. </legal notes>

parameters
=================

*)

METHOD andMaskIsNotEqualTo
VAR_INPUT
	(* current value to check *)
	currentValue	:LWORD;
	(* 2nd operand for bitwise operation *)
	mask			:LWORD;
	(* unexpected result after masking *)
	unexpectedValue	:LWORD;
	(* message if the assertion is false *)
	message			:AssertMessage;
END_VAR
IF ((currentValue AND mask) = unexpectedValue) THEN
	THIS^.assertionWasWrong(message, THIS^.getDebugInfo('andMaskIsNotEqualTo'));
END_IF
END_METHOD

(*

short summary
=================
This assertion method checks if the selected bit of current value
is equal to the expected value

.. <legal notes>

legal notes
=================
| SPDX-FileCopyrightText: © 2022 ekvip automation GmbH <info@ekvip.de>
| SPDX-License-Identifier: Apache-2.0
| For details check: Apache-2.0_

.. _Apache-2.0: https://www.apache.org/licenses/LICENSE-2.0

.. </legal notes>

parameters
=================

*)

METHOD bitXIsEqualTo
VAR_INPUT
	(* current value to check *)
	currentValue	:LWORD;
	(* number of bit to check *)
	number			:BitNumberLWord;
	(* expected value of bit *)
	expectedValue	:BOOL;
	(* message if the assertion is false *)
	message			:AssertMessage;
END_VAR
IF (
	TO_BOOL(
		TO_LWORD(SHL(THIS^.LSB, number))
		AND currentValue
	) <> expectedValue
) THEN
	THIS^.assertionWasWrong(message, THIS^.getDebugInfo('bitXIsEqualTo'));
END_IF
END_METHOD

(*

short summary
=================
This assertion method checks if the selected bit of current value
is not equal to the unexpected value

.. <legal notes>

legal notes
=================
| SPDX-FileCopyrightText: © 2022 ekvip automation GmbH <info@ekvip.de>
| SPDX-License-Identifier: Apache-2.0
| For details check: Apache-2.0_

.. _Apache-2.0: https://www.apache.org/licenses/LICENSE-2.0

.. </legal notes>

parameters
=================

*)

METHOD bitXIsNotEqualTo
VAR_INPUT
	(* current value to check *)
	currentValue	:LWORD;
	(* number of bit to check *)
	number			:BitNumberLWord;
	(* unexpected value of bit *)
	unexpectedValue	:BOOL;
	(* message if the assertion is false *)
	message			:AssertMessage;
END_VAR
IF (
	TO_BOOL(
		TO_LWORD(SHL(THIS^.LSB, number))
		AND currentValue
	) = unexpectedValue
) THEN
	THIS^.assertionWasWrong(message, THIS^.getDebugInfo('bitXIsNotEqualTo'));
END_IF
END_METHOD

(*

short summary
=================
This assertion method checks if the selected bit of current value
is set

.. <legal notes>

legal notes
=================
| SPDX-FileCopyrightText: © 2022 ekvip automation GmbH <info@ekvip.de>
| SPDX-License-Identifier: Apache-2.0
| For details check: Apache-2.0_

.. _Apache-2.0: https://www.apache.org/licenses/LICENSE-2.0

.. </legal notes>

parameters
=================

*)

METHOD bitXIsSet
VAR_INPUT
	(* current value to check *)
	currentValue	:LWORD;
	(* number of bit to check *)
	number			:BitNumberLWord;
	(* message if the assertion is false *)
	message			:AssertMessage;
END_VAR
IF (
	NOT TO_BOOL(
		TO_LWORD(SHL(THIS^.LSB, number))
		AND currentValue
	)
) THEN
	THIS^.assertionWasWrong(message, THIS^.getDebugInfo('bitXIsSet'));
END_IF
END_METHOD

(*

short summary
=================
This assertion method checks if the selected bit of current value
is unset

.. <legal notes>

legal notes
=================
| SPDX-FileCopyrightText: © 2022 ekvip automation GmbH <info@ekvip.de>
| SPDX-License-Identifier: Apache-2.0
| For details check: Apache-2.0_

.. _Apache-2.0: https://www.apache.org/licenses/LICENSE-2.0

.. </legal notes>

parameters
=================

*)

METHOD bitXIsUnset
VAR_INPUT
	(* current value to check *)
	currentValue	:LWORD;
	(* number of bit to check *)
	number			:BitNumberLWord;
	(* message if the assertion is false *)
	message			:AssertMessage;
END_VAR
IF (
	TO_BOOL(
		TO_LWORD(SHL(THIS^.LSB, number))
		AND currentValue
	)
) THEN
	THIS^.assertionWasWrong(message, THIS^.getDebugInfo('bitXIsUnset'));
END_IF
END_METHOD

(*

short summary
=================
This abstract property returns the class name of the concrete object, 
It's for debugging purpose

.. <legal notes>

legal notes
=================
| SPDX-FileCopyrightText: © 2022 ekvip automation GmbH <info@ekvip.de>
| SPDX-License-Identifier: Apache-2.0
| For details check: Apache-2.0_

.. _Apache-2.0: https://www.apache.org/licenses/LICENSE-2.0

.. </legal notes>

*)

PROPERTY className :CNM_AbstractObject.ClassName
GET
className := 'CNM_AssertionInterfaceLib.LWordAssertions';
END_GET
END_PROPERTY

(*

short summary
=================
This assertion method checks if the least significant bit of current value
is equal to the expected value

.. <legal notes>

legal notes
=================
| SPDX-FileCopyrightText: © 2022 ekvip automation GmbH <info@ekvip.de>
| SPDX-License-Identifier: Apache-2.0
| For details check: Apache-2.0_

.. _Apache-2.0: https://www.apache.org/licenses/LICENSE-2.0

.. </legal notes>

parameters
=================

*)

METHOD lsbIsEqualTo
VAR_INPUT
	(* current value to check *)
	currentValue	:LWORD;
	(* expected value of lsb *)
	expectedValue	:BOOL;
	(* message if the assertion is false *)
	message			:AssertMessage;
END_VAR
IF (TO_BOOL(currentValue AND THIS^.LSB) <> expectedValue) THEN
	THIS^.assertionWasWrong(message, THIS^.getDebugInfo('lsbIsEqualTo'));
END_IF
END_METHOD

(*

short summary
=================
This assertion method checks if the least significant bit of current value
is not equal to the unexpected value

.. <legal notes>

legal notes
=================
| SPDX-FileCopyrightText: © 2022 ekvip automation GmbH <info@ekvip.de>
| SPDX-License-Identifier: Apache-2.0
| For details check: Apache-2.0_

.. _Apache-2.0: https://www.apache.org/licenses/LICENSE-2.0

.. </legal notes>

parameters
=================

*)

METHOD lsbIsNotEqualTo
VAR_INPUT
	(* current value to check *)
	currentValue	:LWORD;
	(* unexpected value of lsb *)
	unexpectedValue	:BOOL;
	(* message if the assertion is false *)
	message			:AssertMessage;
END_VAR
IF (TO_BOOL(currentValue AND THIS^.LSB) = unexpectedValue) THEN
	THIS^.assertionWasWrong(message, THIS^.getDebugInfo('lsbIsNotEqualTo'));
END_IF
END_METHOD

(*

short summary
=================
This assertion method checks if the least significant bit of current value
is set

.. <legal notes>

legal notes
=================
| SPDX-FileCopyrightText: © 2022 ekvip automation GmbH <info@ekvip.de>
| SPDX-License-Identifier: Apache-2.0
| For details check: Apache-2.0_

.. _Apache-2.0: https://www.apache.org/licenses/LICENSE-2.0

.. </legal notes>

parameters
=================

*)

METHOD lsbIsSet
VAR_INPUT
	(* current value to check *)
	currentValue	:LWORD;
	(* message if the assertion is false *)
	message			:AssertMessage;
END_VAR
IF (NOT TO_BOOL(currentValue AND THIS^.LSB)) THEN
	THIS^.assertionWasWrong(message, THIS^.getDebugInfo('lsbIsSet'));
END_IF
END_METHOD

(*

short summary
=================
This assertion method checks if the least significant bit of current value
is unset

.. <legal notes>

legal notes
=================
| SPDX-FileCopyrightText: © 2022 ekvip automation GmbH <info@ekvip.de>
| SPDX-License-Identifier: Apache-2.0
| For details check: Apache-2.0_

.. _Apache-2.0: https://www.apache.org/licenses/LICENSE-2.0

.. </legal notes>

parameters
=================

*)

METHOD lsbIsUnset
VAR_INPUT
	(* current value to check *)
	currentValue	:LWORD;
	(* message if the assertion is false *)
	message			:AssertMessage;
END_VAR
IF (TO_BOOL(currentValue AND THIS^.LSB)) THEN
	THIS^.assertionWasWrong(message, THIS^.getDebugInfo('lsbIsUnset'));
END_IF
END_METHOD

(*

short summary
=================
This assertion method checks if the most significant bit of current value
is equal to the expected value

.. <legal notes>

legal notes
=================
| SPDX-FileCopyrightText: © 2022 ekvip automation GmbH <info@ekvip.de>
| SPDX-License-Identifier: Apache-2.0
| For details check: Apache-2.0_

.. _Apache-2.0: https://www.apache.org/licenses/LICENSE-2.0

.. </legal notes>

parameters
=================

*)

METHOD msbIsEqualTo
VAR_INPUT
	(* current value to check *)
	currentValue	:LWORD;
	(* expected value of msb *)
	expectedValue	:BOOL;
	(* message if the assertion is false *)
	message			:AssertMessage;
END_VAR
IF (TO_BOOL(currentValue AND THIS^.MSB) <> expectedValue) THEN
	THIS^.assertionWasWrong(message, THIS^.getDebugInfo('msbIsEqualTo'));
END_IF
END_METHOD

(*

short summary
=================
This assertion method checks if the most significant bit of current value
is not equal to the unexpected value

.. <legal notes>

legal notes
=================
| SPDX-FileCopyrightText: © 2022 ekvip automation GmbH <info@ekvip.de>
| SPDX-License-Identifier: Apache-2.0
| For details check: Apache-2.0_

.. _Apache-2.0: https://www.apache.org/licenses/LICENSE-2.0

.. </legal notes>

parameters
=================

*)

METHOD msbIsNotEqualTo
VAR_INPUT
	(* current value to check *)
	currentValue	:LWORD;
	(* unexpected value of msb *)
	unexpectedValue	:BOOL;
	(* message if the assertion is false *)
	message			:AssertMessage;
END_VAR
IF (TO_BOOL(currentValue AND THIS^.MSB) = unexpectedValue) THEN
	THIS^.assertionWasWrong(message, THIS^.getDebugInfo('msbIsNotEqualTo'));
END_IF
END_METHOD

(*

short summary
=================
This assertion method checks if the most significant bit of current value
is set

.. <legal notes>

legal notes
=================
| SPDX-FileCopyrightText: © 2022 ekvip automation GmbH <info@ekvip.de>
| SPDX-License-Identifier: Apache-2.0
| For details check: Apache-2.0_

.. _Apache-2.0: https://www.apache.org/licenses/LICENSE-2.0

.. </legal notes>

parameters
=================

*)

METHOD msbIsSet
VAR_INPUT
	(* current value to check *)
	currentValue	:LWORD;
	(* message if the assertion is false *)
	message			:AssertMessage;
END_VAR
IF (NOT TO_BOOL(currentValue AND THIS^.MSB)) THEN
	THIS^.assertionWasWrong(message, THIS^.getDebugInfo('msbIsSet'));
END_IF
END_METHOD

(*

short summary
=================
This assertion method checks if the most significant bit of current value
is unset

.. <legal notes>

legal notes
=================
| SPDX-FileCopyrightText: © 2022 ekvip automation GmbH <info@ekvip.de>
| SPDX-License-Identifier: Apache-2.0
| For details check: Apache-2.0_

.. _Apache-2.0: https://www.apache.org/licenses/LICENSE-2.0

.. </legal notes>

parameters
=================

*)

METHOD msbIsUnset
VAR_INPUT
	(* current value to check *)
	currentValue	:LWORD;
	(* message if the assertion is false *)
	message			:AssertMessage;
END_VAR
IF (TO_BOOL(currentValue AND THIS^.MSB)) THEN
	THIS^.assertionWasWrong(message, THIS^.getDebugInfo('msbIsUnset'));
END_IF
END_METHOD

(*

short summary
=================
This assertion method checks if the result current value bitwise ``OR`` mask is equal to the expected value

.. <legal notes>

legal notes
=================
| SPDX-FileCopyrightText: © 2022 ekvip automation GmbH <info@ekvip.de>
| SPDX-License-Identifier: Apache-2.0
| For details check: Apache-2.0_

.. _Apache-2.0: https://www.apache.org/licenses/LICENSE-2.0

.. </legal notes>

parameters
=================

*)

METHOD orMaskIsEqualTo
VAR_INPUT
	(* current value to check *)
	currentValue	:LWORD;
	(* 2nd operand for bitwise operation *)
	mask			:LWORD;
	(* expected result after masking *)
	expectedValue	:LWORD;
	(* message if the assertion is false *)
	message			:AssertMessage;
END_VAR
IF ((currentValue OR mask) <> expectedValue) THEN
	THIS^.assertionWasWrong(message, THIS^.getDebugInfo('orMaskIsEqualTo'));
END_IF
END_METHOD

(*

short summary
=================
This assertion method checks if the result current value bitwise ``OR`` mask 
is not equal to the unexpected value

.. <legal notes>

legal notes
=================
| SPDX-FileCopyrightText: © 2022 ekvip automation GmbH <info@ekvip.de>
| SPDX-License-Identifier: Apache-2.0
| For details check: Apache-2.0_

.. _Apache-2.0: https://www.apache.org/licenses/LICENSE-2.0

.. </legal notes>

parameters
=================

*)

METHOD orMaskIsNotEqualTo
VAR_INPUT
	(* current value to check *)
	currentValue	:LWORD;
	(* 2nd operand for bitwise operation *)
	mask			:LWORD;
	(* unexpected result after masking *)
	unexpectedValue	:LWORD;
	(* message if the assertion is false *)
	message			:AssertMessage;
END_VAR
IF ((currentValue OR mask) = unexpectedValue) THEN
	THIS^.assertionWasWrong(message, THIS^.getDebugInfo('orMaskIsNotEqualTo'));
END_IF
END_METHOD

(*

short summary
=================
This assertion method checks if the current value is equal to the expected value

.. <legal notes>

legal notes
=================
| SPDX-FileCopyrightText: © 2022 ekvip automation GmbH <info@ekvip.de>
| SPDX-License-Identifier: Apache-2.0
| For details check: Apache-2.0_

.. _Apache-2.0: https://www.apache.org/licenses/LICENSE-2.0

.. </legal notes>

parameters
=================

*)

METHOD valueIsEqualTo
VAR_INPUT
	(* current value to check *)
	currentValue	:LWORD;
	(* expected value to compare *)
	expectedValue	:LWORD;
	(* message if the assertion is false *)
	message			:AssertMessage;
END_VAR
IF (currentValue <> expectedValue) THEN
	THIS^.assertionWasWrong(message, THIS^.getDebugInfo('valueIsEqualTo'));
END_IF
END_METHOD

(*

short summary
=================
This assertion method checks if the current value is greater than the less value

.. <legal notes>

legal notes
=================
| SPDX-FileCopyrightText: © 2022 ekvip automation GmbH <info@ekvip.de>
| SPDX-License-Identifier: Apache-2.0
| For details check: Apache-2.0_

.. _Apache-2.0: https://www.apache.org/licenses/LICENSE-2.0

.. </legal notes>

parameters
=================

*)

METHOD valueIsGreaterThan
VAR_INPUT
	(* current value to check *)
	currentValue	:LWORD;
	(* less than lower limit *)
	lessValue		:LWORD;
	(* message if the assertion is false *)
	message			:AssertMessage;
END_VAR
IF (currentValue <= lessValue) THEN
	THIS^.assertionWasWrong(message, THIS^.getDebugInfo('valueIsGreaterThan'));
END_IF
END_METHOD

(*

short summary
=================
This assertion method checks if the current value is inside a limit

.. attention:: 
	limits are included: ``valueIsInRangeOf(3, 3, 3)`` is a true assertion

.. <legal notes>

legal notes
=================
| SPDX-FileCopyrightText: © 2022 ekvip automation GmbH <info@ekvip.de>
| SPDX-License-Identifier: Apache-2.0
| For details check: Apache-2.0_

.. _Apache-2.0: https://www.apache.org/licenses/LICENSE-2.0

.. </legal notes>

parameters
=================

*)

METHOD valueIsInRangeOf
VAR_INPUT
	(* lower limit for the current value *)
	lowerLimit		:LWORD;
	(* current value to check *)
	currentValue	:LWORD;
	(* upper limit for the current value *)
	upperLimit		:LWORD;
	(* message if the assertion is false *)
	message			:AssertMessage;
END_VAR
IF (
	(currentValue < lowerLimit)
	OR (currentValue > upperLimit)
) THEN
	THIS^.assertionWasWrong(message, THIS^.getDebugInfo('valueIsInRangeOf'));
END_IF
END_METHOD

(*

short summary
=================
This assertion method checks if the current value is less than the greater value

.. <legal notes>

legal notes
=================
| SPDX-FileCopyrightText: © 2022 ekvip automation GmbH <info@ekvip.de>
| SPDX-License-Identifier: Apache-2.0
| For details check: Apache-2.0_

.. _Apache-2.0: https://www.apache.org/licenses/LICENSE-2.0

.. </legal notes>

parameters
=================

*)

METHOD valueIsLessThan
VAR_INPUT
	(* current value to check *)
	currentValue	:LWORD;
	(* greater than upper limit *)
	greaterValue	:LWORD;
	(* message if the assertion is false *)
	message			:AssertMessage;
END_VAR
IF (currentValue >= greaterValue) THEN
	THIS^.assertionWasWrong(message, THIS^.getDebugInfo('valueIsLessThan'));
END_IF
END_METHOD

(*

short summary
=================
This assertion method checks if the current value is less than or equal to the maximum value

.. <legal notes>

legal notes
=================
| SPDX-FileCopyrightText: © 2022 ekvip automation GmbH <info@ekvip.de>
| SPDX-License-Identifier: Apache-2.0
| For details check: Apache-2.0_

.. _Apache-2.0: https://www.apache.org/licenses/LICENSE-2.0

.. </legal notes>

parameters
=================

*)

METHOD valueIsMax
VAR_INPUT
	(* current value to check *)
	currentValue	:LWORD;
	(* upper limit for the current value *)
	maximumValue	:LWORD;
	(* message if the assertion is false *)
	message			:AssertMessage;
END_VAR
IF (currentValue > maximumValue) THEN
	THIS^.assertionWasWrong(message, THIS^.getDebugInfo('valueIsMax'));
END_IF
END_METHOD

(*

short summary
=================
This assertion method checks if the current value is greater than or equal to the minimum value

.. <legal notes>

legal notes
=================
| SPDX-FileCopyrightText: © 2022 ekvip automation GmbH <info@ekvip.de>
| SPDX-License-Identifier: Apache-2.0
| For details check: Apache-2.0_

.. _Apache-2.0: https://www.apache.org/licenses/LICENSE-2.0

.. </legal notes>

parameters
=================

*)

METHOD valueIsMin
VAR_INPUT
	(* current value to check *)
	currentValue	:LWORD;
	(* lower limit for the current value *)
	minimumValue	:LWORD;
	(* message if the assertion is false *)
	message			:AssertMessage;
END_VAR
IF (currentValue < minimumValue) THEN
	THIS^.assertionWasWrong(message, THIS^.getDebugInfo('valueIsMin'));
END_IF
END_METHOD

(*

short summary
=================
This assertion method checks if the current value is not equal to the unexpected value

.. <legal notes>

legal notes
=================
| SPDX-FileCopyrightText: © 2022 ekvip automation GmbH <info@ekvip.de>
| SPDX-License-Identifier: Apache-2.0
| For details check: Apache-2.0_

.. _Apache-2.0: https://www.apache.org/licenses/LICENSE-2.0

.. </legal notes>

parameters
=================

*)

METHOD valueIsNotEqualTo
VAR_INPUT
	(* current value to check *)
	currentValue	:LWORD;
	(* unexpected value to compare *)
	unexpectedValue	:LWORD;
	(* message if the assertion is false *)
	message			:AssertMessage;
END_VAR
IF (currentValue = unexpectedValue) THEN
	THIS^.assertionWasWrong(message, THIS^.getDebugInfo('valueIsNotEqualTo'));
END_IF
END_METHOD

(*

short summary
=================
This assertion method checks if the result current value bitwise ``XOR`` mask is equal to the expected value

.. <legal notes>

legal notes
=================
| SPDX-FileCopyrightText: © 2022 ekvip automation GmbH <info@ekvip.de>
| SPDX-License-Identifier: Apache-2.0
| For details check: Apache-2.0_

.. _Apache-2.0: https://www.apache.org/licenses/LICENSE-2.0

.. </legal notes>

parameters
=================

*)

METHOD xorMaskIsEqualTo
VAR_INPUT
	(* current value to check *)
	currentValue	:LWORD;
	(* 2nd operand for bitwise operation *)
	mask			:LWORD;
	(* expected result after masking *)
	expectedValue	:LWORD;
	(* message if the assertion is false *)
	message			:AssertMessage;
END_VAR
IF ((currentValue XOR mask) <> expectedValue) THEN
	THIS^.assertionWasWrong(message, THIS^.getDebugInfo('xorMaskIsEqualTo'));
END_IF
END_METHOD

(*

short summary
=================
This assertion method checks if the result current value bitwise ``XOR`` mask 
is not equal to the unexpected value

.. <legal notes>

legal notes
=================
| SPDX-FileCopyrightText: © 2022 ekvip automation GmbH <info@ekvip.de>
| SPDX-License-Identifier: Apache-2.0
| For details check: Apache-2.0_

.. _Apache-2.0: https://www.apache.org/licenses/LICENSE-2.0

.. </legal notes>

parameters
=================

*)

METHOD xorMaskIsNotEqualTo
VAR_INPUT
	(* current value to check *)
	currentValue	:LWORD;
	(* 2nd operand for bitwise operation *)
	mask			:LWORD;
	(* unexpected result after masking *)
	unexpectedValue	:LWORD;
	(* message if the assertion is false *)
	message			:AssertMessage;
END_VAR
IF ((currentValue XOR mask) = unexpectedValue) THEN
	THIS^.assertionWasWrong(message, THIS^.getDebugInfo('xorMaskIsNotEqualTo'));
END_IF
END_METHOD

END_FUNCTION_BLOCK

// ---- Assertor/Assertions/BitNumberAssertions/XWord/classes/XWordAssertions.TcPOU
(*

short summary
=================
This class provides assert statements for register length words 
It implements :ref:`IXWordAssertions`

.. <legal notes>

legal notes
=================
| SPDX-FileCopyrightText: © 2022 ekvip automation GmbH <info@ekvip.de>
| SPDX-License-Identifier: Apache-2.0
| For details check: Apache-2.0_

.. _Apache-2.0: https://www.apache.org/licenses/LICENSE-2.0

.. </legal notes>

methods and properties
=======================

*)

{attribute 'reflection'}
FUNCTION_BLOCK INTERNAL XWordAssertions EXTENDS AbstactAssertion IMPLEMENTS IXWordAssertions
VAR
END_VAR
VAR CONSTANT
	(* least significant bit *)
	LSB	:__XWORD := 1;
	(* most significant bit *)
	MSB :__XWORD := (SHL(LSB,((SIZEOF(__XWORD)*8)-1)));
END_VAR

(*

short summary
=================
This assertion method checks if the result current value bitwise ``AND`` mask is equal to the expected value

.. <legal notes>

legal notes
=================
| SPDX-FileCopyrightText: © 2022 ekvip automation GmbH <info@ekvip.de>
| SPDX-License-Identifier: Apache-2.0
| For details check: Apache-2.0_

.. _Apache-2.0: https://www.apache.org/licenses/LICENSE-2.0

.. </legal notes>

parameters
=================

*)

METHOD andMaskIsEqualTo
VAR_INPUT
	(* current value to check *)
	currentValue	:__XWORD;
	(* 2nd operand for bitwise operation *)
	mask			:__XWORD;
	(* expected result after masking *)
	expectedValue	:__XWORD;
	(* message if the assertion is false *)
	message			:AssertMessage;
END_VAR
IF ((currentValue AND mask) <> expectedValue) THEN
	THIS^.assertionWasWrong(message, THIS^.getDebugInfo('andMaskIsEqualTo'));
END_IF
END_METHOD

(*

short summary
=================
This assertion method checks if the result current value bitwise ``AND`` mask
is not equal to the unexpected value

.. <legal notes>

legal notes
=================
| SPDX-FileCopyrightText: © 2022 ekvip automation GmbH <info@ekvip.de>
| SPDX-License-Identifier: Apache-2.0
| For details check: Apache-2.0_

.. _Apache-2.0: https://www.apache.org/licenses/LICENSE-2.0

.. </legal notes>

parameters
=================

*)

METHOD andMaskIsNotEqualTo
VAR_INPUT
	(* current value to check *)
	currentValue	:__XWORD;
	(* 2nd operand for bitwise operation *)
	mask			:__XWORD;
	(* unexpected result after masking *)
	unexpectedValue	:__XWORD;
	(* message if the assertion is false *)
	message			:AssertMessage;
END_VAR
IF ((currentValue AND mask) = unexpectedValue) THEN
	THIS^.assertionWasWrong(message, THIS^.getDebugInfo('andMaskIsNotEqualTo'));
END_IF
END_METHOD

(*

short summary
=================
This assertion method checks if the selected bit of current value
is equal to the expected value

.. <legal notes>

legal notes
=================
| SPDX-FileCopyrightText: © 2022 ekvip automation GmbH <info@ekvip.de>
| SPDX-License-Identifier: Apache-2.0
| For details check: Apache-2.0_

.. _Apache-2.0: https://www.apache.org/licenses/LICENSE-2.0

.. </legal notes>

parameters
=================

*)

METHOD bitXIsEqualTo
VAR_INPUT
	(* current value to check *)
	currentValue	:__XWORD;
	(* number of bit to check *)
	number			:BitNumberXWord;
	(* expected value of bit *)
	expectedValue	:BOOL;
	(* message if the assertion is false *)
	message			:AssertMessage;
END_VAR
IF (
	TO_BOOL(
		TO_LWORD(SHL(THIS^.LSB, number))
		AND currentValue
	) <> expectedValue
) THEN
	THIS^.assertionWasWrong(message, THIS^.getDebugInfo('bitXIsEqualTo'));
END_IF
END_METHOD

(*

short summary
=================
This assertion method checks if the selected bit of current value
is not equal to the unexpected value

.. <legal notes>

legal notes
=================
| SPDX-FileCopyrightText: © 2022 ekvip automation GmbH <info@ekvip.de>
| SPDX-License-Identifier: Apache-2.0
| For details check: Apache-2.0_

.. _Apache-2.0: https://www.apache.org/licenses/LICENSE-2.0

.. </legal notes>

parameters
=================

*)

METHOD bitXIsNotEqualTo
VAR_INPUT
	(* current value to check *)
	currentValue	:__XWORD;
	(* number of bit to check *)
	number			:BitNumberXWord;
	(* unexpected value of bit *)
	unexpectedValue	:BOOL;
	(* message if the assertion is false *)
	message			:AssertMessage;
END_VAR
IF (
	TO_BOOL(
		TO_LWORD(SHL(THIS^.LSB, number))
		AND currentValue
	) = unexpectedValue
) THEN
	THIS^.assertionWasWrong(message, THIS^.getDebugInfo('bitXIsNotEqualTo'));
END_IF
END_METHOD

(*

short summary
=================
This assertion method checks if the selected bit of current value
is set

.. <legal notes>

legal notes
=================
| SPDX-FileCopyrightText: © 2022 ekvip automation GmbH <info@ekvip.de>
| SPDX-License-Identifier: Apache-2.0
| For details check: Apache-2.0_

.. _Apache-2.0: https://www.apache.org/licenses/LICENSE-2.0

.. </legal notes>

parameters
=================

*)

METHOD bitXIsSet
VAR_INPUT
	(* current value to check *)
	currentValue	:__XWORD;
	(* number of bit to check *)
	number			:BitNumberXWord;
	(* message if the assertion is false *)
	message			:AssertMessage;
END_VAR
IF (
	NOT TO_BOOL(
		TO_LWORD(SHL(THIS^.LSB, number))
		AND currentValue
	)
) THEN
	THIS^.assertionWasWrong(message, THIS^.getDebugInfo('bitXIsSet'));
END_IF
END_METHOD

(*

short summary
=================
This assertion method checks if the selected bit of current value
is unset

.. <legal notes>

legal notes
=================
| SPDX-FileCopyrightText: © 2022 ekvip automation GmbH <info@ekvip.de>
| SPDX-License-Identifier: Apache-2.0
| For details check: Apache-2.0_

.. _Apache-2.0: https://www.apache.org/licenses/LICENSE-2.0

.. </legal notes>

parameters
=================

*)

METHOD bitXIsUnset
VAR_INPUT
	(* current value to check *)
	currentValue	:__XWORD;
	(* number of bit to check *)
	number			:BitNumberXWord;
	(* message if the assertion is false *)
	message			:AssertMessage;
END_VAR
IF (
	TO_BOOL(
		TO_LWORD(SHL(THIS^.LSB, number))
		AND currentValue
	)
) THEN
	THIS^.assertionWasWrong(message, THIS^.getDebugInfo('bitXIsUnset'));
END_IF
END_METHOD

(*

short summary
=================
This abstract property returns the class name of the concrete object, 
It's for debugging purpose

.. <legal notes>

legal notes
=================
| SPDX-FileCopyrightText: © 2022 ekvip automation GmbH <info@ekvip.de>
| SPDX-License-Identifier: Apache-2.0
| For details check: Apache-2.0_

.. _Apache-2.0: https://www.apache.org/licenses/LICENSE-2.0

.. </legal notes>

*)

PROPERTY className :CNM_AbstractObject.ClassName
GET
className := 'CNM_AssertionInterfaceLib.XWordAssertions';
END_GET
END_PROPERTY

(*

short summary
=================
This assertion method checks if the least significant bit of current value
is equal to the expected value

.. <legal notes>

legal notes
=================
| SPDX-FileCopyrightText: © 2022 ekvip automation GmbH <info@ekvip.de>
| SPDX-License-Identifier: Apache-2.0
| For details check: Apache-2.0_

.. _Apache-2.0: https://www.apache.org/licenses/LICENSE-2.0

.. </legal notes>

parameters
=================

*)

METHOD lsbIsEqualTo
VAR_INPUT
	(* current value to check *)
	currentValue	:__XWORD;
	(* expected value of lsb *)
	expectedValue	:BOOL;
	(* message if the assertion is false *)
	message			:AssertMessage;
END_VAR
IF (TO_BOOL(currentValue AND THIS^.LSB) <> expectedValue) THEN
	THIS^.assertionWasWrong(message, THIS^.getDebugInfo('lsbIsEqualTo'));
END_IF
END_METHOD

(*

short summary
=================
This assertion method checks if the least significant bit of current value
is not equal to the unexpected value

.. <legal notes>

legal notes
=================
| SPDX-FileCopyrightText: © 2022 ekvip automation GmbH <info@ekvip.de>
| SPDX-License-Identifier: Apache-2.0
| For details check: Apache-2.0_

.. _Apache-2.0: https://www.apache.org/licenses/LICENSE-2.0

.. </legal notes>

parameters
=================

*)

METHOD lsbIsNotEqualTo
VAR_INPUT
	(* current value to check *)
	currentValue	:__XWORD;
	(* unexpected value of lsb *)
	unexpectedValue	:BOOL;
	(* message if the assertion is false *)
	message			:AssertMessage;
END_VAR
IF (TO_BOOL(currentValue AND THIS^.LSB) = unexpectedValue) THEN
	THIS^.assertionWasWrong(message, THIS^.getDebugInfo('lsbIsNotEqualTo'));
END_IF
END_METHOD

(*

short summary
=================
This assertion method checks if the least significant bit of current value
is set

.. <legal notes>

legal notes
=================
| SPDX-FileCopyrightText: © 2022 ekvip automation GmbH <info@ekvip.de>
| SPDX-License-Identifier: Apache-2.0
| For details check: Apache-2.0_

.. _Apache-2.0: https://www.apache.org/licenses/LICENSE-2.0

.. </legal notes>

parameters
=================

*)

METHOD lsbIsSet
VAR_INPUT
	(* current value to check *)
	currentValue	:__XWORD;
	(* message if the assertion is false *)
	message			:AssertMessage;
END_VAR
IF (NOT TO_BOOL(currentValue AND THIS^.LSB)) THEN
	THIS^.assertionWasWrong(message, THIS^.getDebugInfo('lsbIsSet'));
END_IF
END_METHOD

(*

short summary
=================
This assertion method checks if the least significant bit of current value
is unset

.. <legal notes>

legal notes
=================
| SPDX-FileCopyrightText: © 2022 ekvip automation GmbH <info@ekvip.de>
| SPDX-License-Identifier: Apache-2.0
| For details check: Apache-2.0_

.. _Apache-2.0: https://www.apache.org/licenses/LICENSE-2.0

.. </legal notes>

parameters
=================

*)

METHOD lsbIsUnset
VAR_INPUT
	(* current value to check *)
	currentValue	:__XWORD;
	(* message if the assertion is false *)
	message			:AssertMessage;
END_VAR
IF (TO_BOOL(currentValue AND THIS^.LSB)) THEN
	THIS^.assertionWasWrong(message, THIS^.getDebugInfo('lsbIsUnset'));
END_IF
END_METHOD

(*

short summary
=================
This assertion method checks if the most significant bit of current value
is equal to the expected value

.. <legal notes>

legal notes
=================
| SPDX-FileCopyrightText: © 2022 ekvip automation GmbH <info@ekvip.de>
| SPDX-License-Identifier: Apache-2.0
| For details check: Apache-2.0_

.. _Apache-2.0: https://www.apache.org/licenses/LICENSE-2.0

.. </legal notes>

parameters
=================

*)

METHOD msbIsEqualTo
VAR_INPUT
	(* current value to check *)
	currentValue	:__XWORD;
	(* expected value of msb *)
	expectedValue	:BOOL;
	(* message if the assertion is false *)
	message			:AssertMessage;
END_VAR
IF (TO_BOOL(currentValue AND THIS^.MSB) <> expectedValue) THEN
	THIS^.assertionWasWrong(message, THIS^.getDebugInfo('msbIsEqualTo'));
END_IF
END_METHOD

(*

short summary
=================
This assertion method checks if the most significant bit of current value
is not equal to the unexpected value

.. <legal notes>

legal notes
=================
| SPDX-FileCopyrightText: © 2022 ekvip automation GmbH <info@ekvip.de>
| SPDX-License-Identifier: Apache-2.0
| For details check: Apache-2.0_

.. _Apache-2.0: https://www.apache.org/licenses/LICENSE-2.0

.. </legal notes>

parameters
=================

*)

METHOD msbIsNotEqualTo
VAR_INPUT
	(* current value to check *)
	currentValue	:__XWORD;
	(* unexpected value of msb *)
	unexpectedValue	:BOOL;
	(* message if the assertion is false *)
	message			:AssertMessage;
END_VAR
IF (TO_BOOL(currentValue AND THIS^.MSB) = unexpectedValue) THEN
	THIS^.assertionWasWrong(message, THIS^.getDebugInfo('msbIsNotEqualTo'));
END_IF
END_METHOD

(*

short summary
=================
This assertion method checks if the most significant bit of current value
is set

.. <legal notes>

legal notes
=================
| SPDX-FileCopyrightText: © 2022 ekvip automation GmbH <info@ekvip.de>
| SPDX-License-Identifier: Apache-2.0
| For details check: Apache-2.0_

.. _Apache-2.0: https://www.apache.org/licenses/LICENSE-2.0

.. </legal notes>

parameters
=================

*)

METHOD msbIsSet
VAR_INPUT
	(* current value to check *)
	currentValue	:__XWORD;
	(* message if the assertion is false *)
	message			:AssertMessage;
END_VAR
IF (NOT TO_BOOL(currentValue AND THIS^.MSB)) THEN
	THIS^.assertionWasWrong(message, THIS^.getDebugInfo('msbIsSet'));
END_IF
END_METHOD

(*

short summary
=================
This assertion method checks if the most significant bit of current value
is unset

.. <legal notes>

legal notes
=================
| SPDX-FileCopyrightText: © 2022 ekvip automation GmbH <info@ekvip.de>
| SPDX-License-Identifier: Apache-2.0
| For details check: Apache-2.0_

.. _Apache-2.0: https://www.apache.org/licenses/LICENSE-2.0

.. </legal notes>

parameters
=================

*)

METHOD msbIsUnset
VAR_INPUT
	(* current value to check *)
	currentValue	:__XWORD;
	(* message if the assertion is false *)
	message			:AssertMessage;
END_VAR
IF (TO_BOOL(currentValue AND THIS^.MSB)) THEN
	THIS^.assertionWasWrong(message, THIS^.getDebugInfo('msbIsUnset'));
END_IF
END_METHOD

(*

short summary
=================
This assertion method checks if the result current value bitwise ``OR`` mask is equal to the expected value

.. <legal notes>

legal notes
=================
| SPDX-FileCopyrightText: © 2022 ekvip automation GmbH <info@ekvip.de>
| SPDX-License-Identifier: Apache-2.0
| For details check: Apache-2.0_

.. _Apache-2.0: https://www.apache.org/licenses/LICENSE-2.0

.. </legal notes>

parameters
=================

*)

METHOD orMaskIsEqualTo
VAR_INPUT
	(* current value to check *)
	currentValue	:__XWORD;
	(* 2nd operand for bitwise operation *)
	mask			:__XWORD;
	(* expected result after masking *)
	expectedValue	:__XWORD;
	(* message if the assertion is false *)
	message			:AssertMessage;
END_VAR
IF ((currentValue OR mask) <> expectedValue) THEN
	THIS^.assertionWasWrong(message, THIS^.getDebugInfo('orMaskIsEqualTo'));
END_IF
END_METHOD

(*

short summary
=================
This assertion method checks if the result current value bitwise ``OR`` mask 
is not equal to the unexpected value

.. <legal notes>

legal notes
=================
| SPDX-FileCopyrightText: © 2022 ekvip automation GmbH <info@ekvip.de>
| SPDX-License-Identifier: Apache-2.0
| For details check: Apache-2.0_

.. _Apache-2.0: https://www.apache.org/licenses/LICENSE-2.0

.. </legal notes>

parameters
=================

*)

METHOD orMaskIsNotEqualTo
VAR_INPUT
	(* current value to check *)
	currentValue	:__XWORD;
	(* 2nd operand for bitwise operation *)
	mask			:__XWORD;
	(* unexpected result after masking *)
	unexpectedValue	:__XWORD;
	(* message if the assertion is false *)
	message			:AssertMessage;
END_VAR
IF ((currentValue OR mask) = unexpectedValue) THEN
	THIS^.assertionWasWrong(message, THIS^.getDebugInfo('orMaskIsNotEqualTo'));
END_IF
END_METHOD

(*

short summary
=================
This assertion method checks if the current value is equal to the expected value

.. <legal notes>

legal notes
=================
| SPDX-FileCopyrightText: © 2022 ekvip automation GmbH <info@ekvip.de>
| SPDX-License-Identifier: Apache-2.0
| For details check: Apache-2.0_

.. _Apache-2.0: https://www.apache.org/licenses/LICENSE-2.0

.. </legal notes>

parameters
=================

*)

METHOD valueIsEqualTo
VAR_INPUT
	(* current value to check *)
	currentValue	:__XWORD;
	(* expected value to compare *)
	expectedValue	:__XWORD;
	(* message if the assertion is false *)
	message			:AssertMessage;
END_VAR
IF (currentValue <> expectedValue) THEN
	THIS^.assertionWasWrong(message, THIS^.getDebugInfo('valueIsEqualTo'));
END_IF
END_METHOD

(*

short summary
=================
This assertion method checks if the current value is greater than the less value

.. <legal notes>

legal notes
=================
| SPDX-FileCopyrightText: © 2022 ekvip automation GmbH <info@ekvip.de>
| SPDX-License-Identifier: Apache-2.0
| For details check: Apache-2.0_

.. _Apache-2.0: https://www.apache.org/licenses/LICENSE-2.0

.. </legal notes>

parameters
=================

*)

METHOD valueIsGreaterThan
VAR_INPUT
	(* current value to check *)
	currentValue	:__XWORD;
	(* less than lower limit *)
	lessValue		:__XWORD;
	(* message if the assertion is false *)
	message			:AssertMessage;
END_VAR
IF (currentValue <= lessValue) THEN
	THIS^.assertionWasWrong(message, THIS^.getDebugInfo('valueIsGreaterThan'));
END_IF
END_METHOD

(*

short summary
=================
This assertion method checks if the current value is inside a limit

.. attention:: 
	limits are included: ``valueIsInRangeOf(3, 3, 3)`` is a true assertion

.. <legal notes>

legal notes
=================
| SPDX-FileCopyrightText: © 2022 ekvip automation GmbH <info@ekvip.de>
| SPDX-License-Identifier: Apache-2.0
| For details check: Apache-2.0_

.. _Apache-2.0: https://www.apache.org/licenses/LICENSE-2.0

.. </legal notes>

parameters
=================

*)

METHOD valueIsInRangeOf
VAR_INPUT
	(* lower limit for the current value *)
	lowerLimit		:__XWORD;
	(* current value to check *)
	currentValue	:__XWORD;
	(* upper limit for the current value *)
	upperLimit		:__XWORD;
	(* message if the assertion is false *)
	message			:AssertMessage;
END_VAR
IF (
	(currentValue < lowerLimit)
	OR (currentValue > upperLimit)
) THEN
	THIS^.assertionWasWrong(message, THIS^.getDebugInfo('valueIsInRangeOf'));
END_IF
END_METHOD

(*

short summary
=================
This assertion method checks if the current value is less than the greater value

.. <legal notes>

legal notes
=================
| SPDX-FileCopyrightText: © 2022 ekvip automation GmbH <info@ekvip.de>
| SPDX-License-Identifier: Apache-2.0
| For details check: Apache-2.0_

.. _Apache-2.0: https://www.apache.org/licenses/LICENSE-2.0

.. </legal notes>

parameters
=================

*)

METHOD valueIsLessThan
VAR_INPUT
	(* current value to check *)
	currentValue	:__XWORD;
	(* greater than upper limit *)
	greaterValue	:__XWORD;
	(* message if the assertion is false *)
	message			:AssertMessage;
END_VAR
IF (currentValue >= greaterValue) THEN
	THIS^.assertionWasWrong(message, THIS^.getDebugInfo('valueIsLessThan'));
END_IF
END_METHOD

(*

short summary
=================
This assertion method checks if the current value is less than or equal to the maximum value

.. <legal notes>

legal notes
=================
| SPDX-FileCopyrightText: © 2022 ekvip automation GmbH <info@ekvip.de>
| SPDX-License-Identifier: Apache-2.0
| For details check: Apache-2.0_

.. _Apache-2.0: https://www.apache.org/licenses/LICENSE-2.0

.. </legal notes>

parameters
=================

*)

METHOD valueIsMax
VAR_INPUT
	(* current value to check *)
	currentValue	:__XWORD;
	(* upper limit for the current value *)
	maximumValue	:__XWORD;
	(* message if the assertion is false *)
	message			:AssertMessage;
END_VAR
IF (currentValue > maximumValue) THEN
	THIS^.assertionWasWrong(message, THIS^.getDebugInfo('valueIsMax'));
END_IF
END_METHOD

(*

short summary
=================
This assertion method checks if the current value is greater than or equal to the minimum value

.. <legal notes>

legal notes
=================
| SPDX-FileCopyrightText: © 2022 ekvip automation GmbH <info@ekvip.de>
| SPDX-License-Identifier: Apache-2.0
| For details check: Apache-2.0_

.. _Apache-2.0: https://www.apache.org/licenses/LICENSE-2.0

.. </legal notes>

parameters
=================

*)

METHOD valueIsMin
VAR_INPUT
	(* current value to check *)
	currentValue	:__XWORD;
	(* lower limit for the current value *)
	minimumValue	:__XWORD;
	(* message if the assertion is false *)
	message			:AssertMessage;
END_VAR
IF (currentValue < minimumValue) THEN
	THIS^.assertionWasWrong(message, THIS^.getDebugInfo('valueIsMin'));
END_IF
END_METHOD

(*

short summary
=================
This assertion method checks if the current value is not equal to the unexpected value

.. <legal notes>

legal notes
=================
| SPDX-FileCopyrightText: © 2022 ekvip automation GmbH <info@ekvip.de>
| SPDX-License-Identifier: Apache-2.0
| For details check: Apache-2.0_

.. _Apache-2.0: https://www.apache.org/licenses/LICENSE-2.0

.. </legal notes>

parameters
=================

*)

METHOD valueIsNotEqualTo
VAR_INPUT
	(* current value to check *)
	currentValue	:__XWORD;
	(* unexpected value to compare *)
	unexpectedValue	:__XWORD;
	(* message if the assertion is false *)
	message			:AssertMessage;
END_VAR
IF (currentValue = unexpectedValue) THEN
	THIS^.assertionWasWrong(message, THIS^.getDebugInfo('valueIsNotEqualTo'));
END_IF
END_METHOD

(*

short summary
=================
This assertion method checks if the result current value bitwise ``XOR`` mask is equal to the expected value

.. <legal notes>

legal notes
=================
| SPDX-FileCopyrightText: © 2022 ekvip automation GmbH <info@ekvip.de>
| SPDX-License-Identifier: Apache-2.0
| For details check: Apache-2.0_

.. _Apache-2.0: https://www.apache.org/licenses/LICENSE-2.0

.. </legal notes>

parameters
=================

*)

METHOD xorMaskIsEqualTo
VAR_INPUT
	(* current value to check *)
	currentValue	:__XWORD;
	(* 2nd operand for bitwise operation *)
	mask			:__XWORD;
	(* expected result after masking *)
	expectedValue	:__XWORD;
	(* message if the assertion is false *)
	message			:AssertMessage;
END_VAR
IF ((currentValue XOR mask) <> expectedValue) THEN
	THIS^.assertionWasWrong(message, THIS^.getDebugInfo('xorMaskIsEqualTo'));
END_IF
END_METHOD

(*

short summary
=================
This assertion method checks if the result current value bitwise ``XOR`` mask 
is not equal to the unexpected value

.. <legal notes>

legal notes
=================
| SPDX-FileCopyrightText: © 2022 ekvip automation GmbH <info@ekvip.de>
| SPDX-License-Identifier: Apache-2.0
| For details check: Apache-2.0_

.. _Apache-2.0: https://www.apache.org/licenses/LICENSE-2.0

.. </legal notes>

parameters
=================

*)

METHOD xorMaskIsNotEqualTo
VAR_INPUT
	(* current value to check *)
	currentValue	:__XWORD;
	(* 2nd operand for bitwise operation *)
	mask			:__XWORD;
	(* unexpected result after masking *)
	unexpectedValue	:__XWORD;
	(* message if the assertion is false *)
	message			:AssertMessage;
END_VAR
IF ((currentValue XOR mask) = unexpectedValue) THEN
	THIS^.assertionWasWrong(message, THIS^.getDebugInfo('xorMaskIsNotEqualTo'));
END_IF
END_METHOD

END_FUNCTION_BLOCK

// ---- Assertor/Assertions/BooleanAssertion/classes/BooleanAssertion.TcPOU
(*

short summary
=================
This class provides assert statements for booleans.
It implements the interface :ref:`IBooleanAssertion`

.. <legal notes>

legal notes
=================
| SPDX-FileCopyrightText: © 2022 ekvip automation GmbH <info@ekvip.de>
| SPDX-License-Identifier: Apache-2.0
| For details check: Apache-2.0_

.. _Apache-2.0: https://www.apache.org/licenses/LICENSE-2.0

.. </legal notes>

methods and properties
==================

*)

{attribute 'reflection'}
FUNCTION_BLOCK INTERNAL BooleanAssertion EXTENDS AbstactAssertion IMPLEMENTS IBooleanAssertion
VAR
END_VAR

(*

short summary
=================
This abstract property returns the class name of the concrete object, 
It's for debugging purpose

.. <legal notes>

legal notes
=================
| SPDX-FileCopyrightText: © 2022 ekvip automation GmbH <info@ekvip.de>
| SPDX-License-Identifier: Apache-2.0
| For details check: Apache-2.0_

.. _Apache-2.0: https://www.apache.org/licenses/LICENSE-2.0

.. </legal notes>

*)

PROPERTY className :CNM_AbstractObject.ClassName
GET
className := 'CNM_AssertionInterfaceLib.BooleanAssertion';
END_GET
END_PROPERTY

(*

short summary
=================
This assertion method checks if the current value is equal to the expected value

.. <legal notes>

legal notes
=================
| SPDX-FileCopyrightText: © 2022 ekvip automation GmbH <info@ekvip.de>
| SPDX-License-Identifier: Apache-2.0
| For details check: Apache-2.0_

.. _Apache-2.0: https://www.apache.org/licenses/LICENSE-2.0

.. </legal notes>

parameters
=================

*)

METHOD valueIsEqualTo
VAR_INPUT
	(* current value to check *)
	currentValue	:BOOL;
	(* expected value to compare *)
	expectedValue	:BOOL;
	(* message if the assertion is false *)
	message			:AssertMessage;
END_VAR
IF (currentValue <> expectedValue) THEN	
	THIS^.assertionWasWrong(message, THIS^.getDebugInfo('valueIsEqualTo'));
END_IF
END_METHOD

(*

short summary
=================
This assertion method checks if the current value is ``FALSE``

.. <legal notes>

legal notes
=================
| SPDX-FileCopyrightText: © 2022 ekvip automation GmbH <info@ekvip.de>
| SPDX-License-Identifier: Apache-2.0
| For details check: Apache-2.0_

.. _Apache-2.0: https://www.apache.org/licenses/LICENSE-2.0

.. </legal notes>

parameters
=================

*)

METHOD valueIsFalse
VAR_INPUT
	(* current value to check *)
	currentValue	:BOOL;
	(* message if the assertion is false *)
	message	: AssertMessage;
END_VAR
IF (currentValue) THEN
	THIS^.assertionWasWrong(message, THIS^.getDebugInfo('valueIsFalse'));
END_IF
END_METHOD

(*

short summary
=================
This assertion method checks if the current value is not equal to the unexpected value

.. <legal notes>

legal notes
=================
| SPDX-FileCopyrightText: © 2022 ekvip automation GmbH <info@ekvip.de>
| SPDX-License-Identifier: Apache-2.0
| For details check: Apache-2.0_

.. _Apache-2.0: https://www.apache.org/licenses/LICENSE-2.0

.. </legal notes>

parameters
=================

*)

METHOD valueIsNotEqualTo
VAR_INPUT
	(* current value to check *)
	currentValue	:BOOL;
	(* unexpected value to compare *)
	unexpectedValue	:BOOL;
	(* message if the assertion is false *)
	message			:AssertMessage;
END_VAR
IF (currentValue = unexpectedValue) THEN	
	THIS^.assertionWasWrong(message, THIS^.getDebugInfo('valueIsNotEqualTo'));
END_IF
END_METHOD

(*

short summary
=================
This assertion method checks if the current value is ``TRUE``

.. <legal notes>

legal notes
=================
| SPDX-FileCopyrightText: © 2022 ekvip automation GmbH <info@ekvip.de>
| SPDX-License-Identifier: Apache-2.0
| For details check: Apache-2.0_

.. _Apache-2.0: https://www.apache.org/licenses/LICENSE-2.0

.. </legal notes>

parameters
=================

*)

METHOD valueIsTrue
VAR_INPUT
	(* current value to check *)
	currentValue	:BOOL;
	(* message if the assertion is false *)
	message	: AssertMessage;
END_VAR
IF (NOT currentValue) THEN
	THIS^.assertionWasWrong(message, THIS^.getDebugInfo('valueIsTrue'));
END_IF
END_METHOD

END_FUNCTION_BLOCK

// ---- Assertor/Assertions/classes/Assertions.TcPOU
(*

short summary
=================
| This class provides assert statements the most common data:
| It implements the interface :ref:`IAssertions`
| For ``STRUCT``, ``ARRAY``, ``FUNCTION BLOCK``, ``ENUM``  use :ref:`Assertions.binary`
| For ``BYTE``, ``WORD``, ``DWORD``, ``LWORD``, ``__XWORD`` use :ref:`Assertions.bitNumber`
| For ``BOOL`` use :ref:`Assertions.boolean`
| For ``DT``, ``TOD``, ``DATE`` use :ref:`Assertions.dateAndTime`
| For ``REAL``, ``LREAL`` use :ref:`Assertions.float`
| For ``SINT``, ``INT``, ``DINT``, ``LINT``, ``__XINT`` use :ref:`Assertions.integer`
| For ``CNM_AbsrtractObject.IObject`` use :ref:`Assertions.object`
| For ``POINTER`` use :ref:`Assertions.pointers`
| For ``STRING``, ``WSTRING`` use :ref:`Assertions.strings`
| For ``TIME``, ``LTIME`` use :ref:`Assertions.times`

.. <legal notes>

legal notes
=================
| SPDX-FileCopyrightText: © 2022 ekvip automation GmbH <info@ekvip.de>
| SPDX-License-Identifier: Apache-2.0
| For details check: Apache-2.0_

.. _Apache-2.0: https://www.apache.org/licenses/LICENSE-2.0

.. </legal notes>

methods and properties
=======================

*)

{attribute 'reflection'}
FUNCTION_BLOCK INTERNAL Assertions EXTENDS CNM_AbstractObject.Object IMPLEMENTS IAssertions, IAssertCallBacksetter
VAR
	(* class to handle binary assertions *)
	binaryAssertions	:BinaryAssertions();
	(* class to handle bit number assertions *)
	bitNumberAssertions	:BitNumberAssertions();
	(* class to handle boolean assertions *)
	booleanAssertions	:BooleanAssertion();
	(* class to handle date and time assertions *)
	dateTimeAssertions	:DateAndTimeAssertions();
	(* class to handle float assertions *)
	floatAssertions		:FloatAssertions();
	(* class to handle integer assertions *)
	intgerAssertions	:IntergerAssertions();
	(* class to handle object assertions *)
	objectAssertions	:ObjectAssertions();
	(* class to handle pointer assertions *)
	pointerAssertions	:PointerAssertions();
	(* class to handle string assertions *)
	stringAssertions	:StringAssertions();
	(* class to handle time assertions *)
	timeAssertions		:TimeAssertions();
END_VAR

(*

short summary
=================
Returns the interface :ref:`IBinaryAssertions`
with assert statements for binary data 

.. <legal notes>

legal notes
=================
| SPDX-FileCopyrightText: © 2022 ekvip automation GmbH <info@ekvip.de>
| SPDX-License-Identifier: Apache-2.0
| For details check: Apache-2.0_

.. _Apache-2.0: https://www.apache.org/licenses/LICENSE-2.0

.. </legal notes>

*)

PROPERTY binary :IBinaryAssertions
GET
binary := THIS^.binaryAssertions;
END_GET
END_PROPERTY

(*

short summary
=================
Returns the interface :ref:`IBitNumberAssertions`
with assert statements for bit numbers 

.. <legal notes>

legal notes
=================
| SPDX-FileCopyrightText: © 2022 ekvip automation GmbH <info@ekvip.de>
| SPDX-License-Identifier: Apache-2.0
| For details check: Apache-2.0_

.. _Apache-2.0: https://www.apache.org/licenses/LICENSE-2.0

.. </legal notes>

*)

PROPERTY bitNumber :IBitNumberAssertions
GET
bitNumber := THIS^.bitNumberAssertions;
END_GET
END_PROPERTY

(*

short summary
=================
Returns the interface :ref:`IBooleanAssertion`
with assert statements for booleans

.. <legal notes>

legal notes
=================
| SPDX-FileCopyrightText: © 2022 ekvip automation GmbH <info@ekvip.de>
| SPDX-License-Identifier: Apache-2.0
| For details check: Apache-2.0_

.. _Apache-2.0: https://www.apache.org/licenses/LICENSE-2.0

.. </legal notes>

*)

PROPERTY boolean :IBooleanAssertion
GET
boolean := THIS^.booleanAssertions;
END_GET
END_PROPERTY

(*

short summary
=================
This abstract property returns the class name of the concrete object, 
It's for debugging purpose

.. <legal notes>

legal notes
=================
| SPDX-FileCopyrightText: © 2022 ekvip automation GmbH <info@ekvip.de>
| SPDX-License-Identifier: Apache-2.0
| For details check: Apache-2.0_

.. _Apache-2.0: https://www.apache.org/licenses/LICENSE-2.0

.. </legal notes>

*)

PROPERTY className :CNM_AbstractObject.ClassName
GET
className := 'CNM_AssertionInterfaceLib.Assertions';
END_GET
END_PROPERTY

(*

short summary
=================
Returns the interface :ref:`IDateAndTimeAssertions`
with assert statements for date and time data types

.. <legal notes>

legal notes
=================
| SPDX-FileCopyrightText: © 2022 ekvip automation GmbH <info@ekvip.de>
| SPDX-License-Identifier: Apache-2.0
| For details check: Apache-2.0_

.. _Apache-2.0: https://www.apache.org/licenses/LICENSE-2.0

.. </legal notes>

*)

PROPERTY dateAndTime :IDateAndTimeAssertions
GET
dateAndTime := THIS^.dateTimeAssertions;
END_GET
END_PROPERTY

(*

short summary
=================
Returns the interface :ref:`IFloatAssertions`
with assert statements for floatings

.. <legal notes>

legal notes
=================
| SPDX-FileCopyrightText: © 2022 ekvip automation GmbH <info@ekvip.de>
| SPDX-License-Identifier: Apache-2.0
| For details check: Apache-2.0_

.. _Apache-2.0: https://www.apache.org/licenses/LICENSE-2.0

.. </legal notes>

*)

PROPERTY float :IFloatAssertions
GET
float := THIS^.floatAssertions;
END_GET
END_PROPERTY

(*

short summary
=================
Returns the interface :ref:`IIntergerAssertions`
with assert statements for integers

.. <legal notes>

legal notes
=================
| SPDX-FileCopyrightText: © 2022 ekvip automation GmbH <info@ekvip.de>
| SPDX-License-Identifier: Apache-2.0
| For details check: Apache-2.0_

.. _Apache-2.0: https://www.apache.org/licenses/LICENSE-2.0

.. </legal notes>

*)

PROPERTY integer :IIntergerAssertions
GET
integer := THIS^.intgerAssertions;
END_GET
END_PROPERTY

(*

short summary
=================
Returns the interface :ref:`IObjectAssertions`
with assert statements for ``CNM_AbstractObject.IObject``

.. <legal notes>

legal notes
=================
| SPDX-FileCopyrightText: © 2022 ekvip automation GmbH <info@ekvip.de>
| SPDX-License-Identifier: Apache-2.0
| For details check: Apache-2.0_

.. _Apache-2.0: https://www.apache.org/licenses/LICENSE-2.0

.. </legal notes>

*)

PROPERTY object :IObjectAssertions
GET
object := THIS^.objectAssertions;
END_GET
END_PROPERTY

(*

short summary
=================
Returns the interface :ref:`IPointerAssertions`
with assert statements for pointers

.. <legal notes>

legal notes
=================
| SPDX-FileCopyrightText: © 2022 ekvip automation GmbH <info@ekvip.de>
| SPDX-License-Identifier: Apache-2.0
| For details check: Apache-2.0_

.. _Apache-2.0: https://www.apache.org/licenses/LICENSE-2.0

.. </legal notes>

*)

PROPERTY pointers :IPointerAssertions
GET
pointers := THIS^.pointerAssertions;
END_GET
END_PROPERTY

(*

short summary
=================
This methods is the setter for the callback class if an assertion was false

.. <legal notes>

legal notes
=================
| SPDX-FileCopyrightText: © 2022 ekvip automation GmbH <info@ekvip.de>
| SPDX-License-Identifier: Apache-2.0
| For details check: Apache-2.0_

.. _Apache-2.0: https://www.apache.org/licenses/LICENSE-2.0

.. </legal notes>

parameters
=================

*)

METHOD setCallBack
VAR_INPUT
	(* the class that must be informed if an assertion is false *)
	callBack	:IAssertCallback;  
END_VAR
THIS^.binaryAssertions.setCallBack(callBack);
THIS^.bitNumberAssertions.setCallBack(callBack);
THIS^.booleanAssertions.setCallBack(callBack);
THIS^.dateTimeAssertions.setCallBack(callBack);
THIS^.floatAssertions.setCallBack(callBack);
THIS^.intgerAssertions.setCallBack(callBack);
THIS^.objectAssertions.setCallBack(callBack);
THIS^.pointerAssertions.setCallBack(callBack);
THIS^.stringAssertions.setCallBack(callBack);
THIS^.timeAssertions.setCallBack(callBack);
END_METHOD

(*

short summary
=================
Returns the interface :ref:`IStringAssertions`
with assert statements for windows-1252 and UTF-16 strings

.. <legal notes>

legal notes
=================
| SPDX-FileCopyrightText: © 2022 ekvip automation GmbH <info@ekvip.de>
| SPDX-License-Identifier: Apache-2.0
| For details check: Apache-2.0_

.. _Apache-2.0: https://www.apache.org/licenses/LICENSE-2.0

.. </legal notes>

*)

PROPERTY strings :IStringAssertions
GET
strings := THIS^.stringAssertions;
END_GET
END_PROPERTY

(*

short summary
=================
Returns the interface :ref:`ITimeAssertions`
with assert statements for time data types

.. <legal notes>

legal notes
=================
| SPDX-FileCopyrightText: © 2022 ekvip automation GmbH <info@ekvip.de>
| SPDX-License-Identifier: Apache-2.0
| For details check: Apache-2.0_

.. _Apache-2.0: https://www.apache.org/licenses/LICENSE-2.0

.. </legal notes>

*)

PROPERTY times :ITimeAssertions
GET
times := THIS^.timeAssertions;
END_GET
END_PROPERTY

END_FUNCTION_BLOCK

// ---- Assertor/Assertions/DateAndTimeAssertions/classes/DateAndTimeAssertions.TcPOU
(*

short summary
=================
| This class provides assert statements for date and time types
| It implements :ref:`IDateAndTimeAssertions`
| For 32 bit date and time types use :ref:`DateAndTimeAssertions.simple`

.. <legal notes>

legal notes
=================
| SPDX-FileCopyrightText: © 2022 ekvip automation GmbH <info@ekvip.de>
| SPDX-License-Identifier: Apache-2.0
| For details check: Apache-2.0_

.. _Apache-2.0: https://www.apache.org/licenses/LICENSE-2.0

.. </legal notes>

methods and properties
=======================

*)

{attribute 'reflection'}
FUNCTION_BLOCK INTERNAL DateAndTimeAssertions
EXTENDS CNM_AbstractObject.Object
IMPLEMENTS IDateAndTimeAssertions, IAssertCallBacksetter
VAR
	(* class to handle 32 bit date and time assertions *)
	assertionsFor32BitTypes	:SimpleDateAndTimeAssertions();
	(* class to handle 64 bit date and time assertions *)
	assertionsFor64BitTypes	:LongDateAndTimeAssertions();
END_VAR

(*

short summary
=================
This abstract property returns the class name of the concrete object, 
It's for debugging purpose

.. <legal notes>

legal notes
=================
| SPDX-FileCopyrightText: © 2022 ekvip automation GmbH <info@ekvip.de>
| SPDX-License-Identifier: Apache-2.0
| For details check: Apache-2.0_

.. _Apache-2.0: https://www.apache.org/licenses/LICENSE-2.0

.. </legal notes>

*)

PROPERTY className :CNM_AbstractObject.ClassName
GET
className := 'CNM_AssertionInterfaceLib.DateAndTimeAssertions';
END_GET
END_PROPERTY

(*

short summary
=================
Returns an interface with assert statements for 64 bit times 

.. <legal notes>

legal notes
=================
| SPDX-FileCopyrightText: © 2022 ekvip automation GmbH <info@ekvip.de>
| SPDX-License-Identifier: Apache-2.0
| For details check: Apache-2.0_

.. _Apache-2.0: https://www.apache.org/licenses/LICENSE-2.0

.. </legal notes>

*)

PROPERTY long :ILongDateAndTimeAssertions
GET
long := THIS^.assertionsFor64BitTypes;
END_GET
END_PROPERTY

(*

short summary
=================
This methods is the setter for the callback class if an assertion was false

.. <legal notes>

legal notes
=================
| SPDX-FileCopyrightText: © 2022 ekvip automation GmbH <info@ekvip.de>
| SPDX-License-Identifier: Apache-2.0
| For details check: Apache-2.0_

.. _Apache-2.0: https://www.apache.org/licenses/LICENSE-2.0

.. </legal notes>

parameters
=================

*)

METHOD setCallBack
VAR_INPUT
	(* the class that must be informed if an assertion is false *)
	callBack	:IAssertCallback;  
END_VAR
THIS^.assertionsFor32BitTypes.setCallBack(callBack);
THIS^.assertionsFor64BitTypes.setCallBack(callBack);
END_METHOD

(*

